# B&R Automation Studio project A2019059_Linka_Power_CP (part 20)

#### Main.st - Init, cyclic, exit code
```iecst
PROGRAM _INIT
    TprazdnyZasobnik.PT:=T#2000ms;
    TakumulaciaPlna.PT:=T#1000ms;
    TvytvorenieVakua.PT:=T#200ms;
    TodvetranieVakua.PT:=T#1s;
    TprefukPredBrzdou.PT:=T#2000ms;
    TprefukZaBrzdou.PT:=T#2000ms;
    TvysuvanieSpindle.PT:=T#1s;
    TpripravaSkrutky.PT:=T#3000ms;
    ToddelovacZakladnaPoloha.PT:=T#1000ms;
    TodsatieNecistot.PT:=T#1000ms;
    Tvibrovanie.PT:=T#3000ms;
    TvyfukovaniePredVibrovanim.PT:= T#1000ms;
    TpodaniaSkrutky.PT:= T#1000ms;
    TpredSkrutkaPripravena.PT:= T#500ms;
    TvypnutieOfuku.PT:= T#2000ms;
    TalarmuVysunutiaSkrutkovacky.PT:= T#10s;
END_PROGRAM

PROGRAM _CYCLIC

	(********************Mapovanie IN/OUT********************************)

    SkrutkovaciSet.Manual:= P1_Srobovanie.SkrutkovaciSet_K30.Manual;
    SkrutkovaciSet.Automat:= P1_Srobovanie.SkrutkovaciSet_K30.Automat;
    SkrutkovaciSet.SkrutkaOdobrata:=P1_Srobovanie.SkrutkovaciSet_K30.SkrutkaK30_Odobrata;
    P1_Srobovanie.SkrutkovaciSet_K30.SkrutkaK30_Pripravena:= SkrutkovaciSet.SkrutkaPripravena;
    P1_Srobovanie.SkrutkovaciSet_K30.CistenieUkoncene:= SkrutkovaciSet.CistenieVykonane;
    SkrutkovaciSet.VykonajCistenie:= P1_Srobovanie.SkrutkovaciSet_K30.Cistenie;

    SkrutkovaciSet.Vreteno.IN.BrakeClosed:=P1_Srobovanie.IN.SkrutkK30_Cist_BrzdaZatvor_MS22;
    SkrutkovaciSet.Vreteno.IN.BrakeOpen:=P1_Srobovanie.IN.SkrutkK30_Cist_BrzdaOtvoren_MS21;
    SkrutkovaciSet.Vreteno.IN.DeptControl:=P1_Srobovanie.IN.SkrutkK30_ZASUNUTY_MS20;
    SkrutkovaciSet.Vreteno.IN.ScrewMeasurement:=P1_Srobovanie.IN.SkrutkK30_SrobaPresla_IS51;
    SkrutkovaciSet.Vreteno.IN.ScrewMeasurementBrake:=P1_Srobovanie.IN.SkrutkK30_Cist_SrobaPresla_IS52;

    IF P1_Srobovanie.SkrutkovaciSet_K30.Reset AND SkrutkovaciSet.VretenoFaza <> 102 AND SkrutkovaciSet.VretenoFaza <> 104 THEN
        SkrutkovaciSet.VretenoFaza:=0;
        P1_Srobovanie.SkrutkovaciSet_K30.Reset:= FALSE;
    END_IF

    SkrutkovaciSet.Zasobnik.IN.AccumulationSwitch:=P1_Srobovanie.IN.ZasobSrobK30_ListaPLNA_OS7;
    SkrutkovaciSet.Zasobnik.IN.FeederLevelControl:=P1_Srobovanie.IN.ZasobSrobK30_PRAZDNY_IS49;
    SkrutkovaciSet.Zasobnik.IN.ScrewMeasurement:=P1_Srobovanie.IN.NastrelSrobK30_SrobaPresla_IS50;

    P1_Srobovanie.OUT.SkrutkK30_Cist_POSUN_YV123:=SkrutkovaciSet.Vreteno.OUT.BlastAirBrake;
    P1_Srobovanie.OUT.SkrutkK30_Cist_OTVOR_YV92:=SkrutkovaciSet.Vreteno.OUT.BrakeSpindle;
    P1_Srobovanie.OUT.SkrutkK30_OfukVakua_RUN_YV91:=SkrutkovaciSet.Vreteno.OUT.CounterBlast;
    IF SkrutkovaciSet.VretenoFaza>1 AND SkrutkovaciSet.VretenoFaza<100 THEN
        P1_Srobovanie.OUT.SkrutkK30_VYSUN_YV89:=SkrutkovaciSet.Vreteno.OUT.Spindle;
    END_IF
    P1_Srobovanie.OUT.SkrutkK30_Cist_ODSAVANIE_YV93:=SkrutkovaciSet.Vreteno.OUT.WasteExtraction;
    IF SkrutkovaciSet.VykonajCistenie THEN
        P1_Srobovanie.OUT.SkrutkK30_PrisavSkrutky_RUN_YV90:=SkrutkovaciSet.Vreteno.OUT.Vacuum;
    END_IF
    P1_Srobovanie.OUT.ZasobSrobK30_Ofuk_RUN_YV85:=SkrutkovaciSet.Zasobnik.OUT.BlowOff;
    P1_Srobovanie.OUT.NastrelSrobK30_PosunSrobu_YV87:=SkrutkovaciSet.Zasobnik.OUT.Escapement;
    P1_Srobovanie.OUT.NastrelSrobK30_NastrelSrobu_YV88:=SkrutkovaciSet.Zasobnik.OUT.FeedAir;
    P1_Srobovanie.OUT.ZasobSrobK30_OfukTried_RUN_YV86:=SkrutkovaciSet.Zasobnik.OUT.SortingAir;
    P1_Srobovanie.OUT.ZasobSrobK30_Vibrovanie_RUN_FM8:= SkrutkovaciSet.Zasobnik.OUT.StartA20;
    (********************Časáky********************************)
    TprazdnyZasobnik();
    TakumulaciaPlna();
    TvytvorenieVakua();
    TodvetranieVakua();
    TprefukPredBrzdou();
    TprefukZaBrzdou();
    TvysuvanieSpindle();
    TpripravaSkrutky();
    ToddelovacZakladnaPoloha();
    TodsatieNecistot();
    Tvibrovanie();
    TvyfukovaniePredVibrovanim();
    TpodaniaSkrutky();
    TpredSkrutkaPripravena();
    TvypnutieOfuku();
    TalarmuVysunutiaSkrutkovacky();
    (********************Zásobnik********************************)

    //kontrola akumulacie
    IF SkrutkovaciSet.Zasobnik.IN.AccumulationSwitch=1 THEN
        TakumulaciaPlna.IN:=1;
    ELSE
        TakumulaciaPlna.IN:=0;
    END_IF

    //kontrola naplnenia zasobnika
    IF SkrutkovaciSet.Zasobnik.IN.FeederLevelControl=1 THEN
        TprazdnyZasobnik.IN:=1;
    ELSE
        TprazdnyZasobnik.IN:=0;
    END_IF

    //Ovládanie vzduchov zásobníka//
    IF ZapniHrniec THEN
        IF TakumulaciaPlna.Q=1 THEN
            SkrutkovaciSet.Zasobnik.OUT.BlowOff:=1;
        ELSE
            SkrutkovaciSet.Zasobnik.OUT.BlowOff:=0;
        END_IF
        SkrutkovaciSet.Zasobnik.OUT.SortingAir:= 1;
    ELSE
        SkrutkovaciSet.Zasobnik.OUT.BlowOff:=0;
    END_IF

    IF NOT SkrutkovaciSet.Zasobnik.OUT.StartA20 AND NOT ZapniHrniec THEN
        TvypnutieOfuku.IN:= 1;
    ELSE
        TvypnutieOfuku.IN:= 0;
    END_IF

    IF EDGEPOS(TvypnutieOfuku.Q) THEN
        SkrutkovaciSet.Zasobnik.OUT.SortingAir:= 0;
    END_IF

    //ovladanie vibracneho podavaca
    IF ZapniHrniec THEN
        TvyfukovaniePredVibrovanim.IN:= 1;
    ELSE
        TvyfukovaniePredVibrovanim.IN:= 0;
    END_IF

    IF ZapniHrniec AND TvyfukovaniePredVibrovanim.Q THEN
        SkrutkovaciSet.Zasobnik.OUT.StartA20:=1;
        Tvibrovanie.IN:=1;
    ELSE
        SkrutkovaciSet.Zasobnik.OUT.StartA20:=0;
        Tvibrovanie.IN:=0;
    END_IF

    IF Tvibrovanie.Q=1 AND NOT P1_Srobovanie.RR_ZapniHrniec_K30 THEN
        IF TakumulaciaPlna.Q=1 THEN
            ZapniHrniec:= 0;
        END_IF
    END_IF

    //Zapnutie hrnca v ručnom režime//
    IF EDGEPOS(P1_Srobovanie.RR_ZapniHrniec_K30) THEN
        ZapniHrniec:= TRUE;
    END_IF
    IF EDGENEG(P1_Srobovanie.RR_ZapniHrniec_K30) THEN
        ZapniHrniec:= FALSE;
    END_IF

    //Zrušenie signálu skrutka pripravená//
    IF SkrutkovaciSet.SkrutkaPripravena=1 THEN
        IF SkrutkovaciSet.SkrutkaOdobrata=1 THEN
            SkrutkovaciSet.SkrutkaPripravena:=0;
        END_IF
    END_IF

    (********************Vreteno********************************)
    CASE SkrutkovaciSet.VretenoFaza OF
        0: SkrutkovaciSet.VretenoStatus:="Vypnute";
            SkrutkovaciSet.Vreteno.OUT.BlastAirBrake:=0;
            SkrutkovaciSet.Vreteno.OUT.BrakeSpindle:=0;
            SkrutkovaciSet.Vreteno.OUT.CounterBlast:=0;
            SkrutkovaciSet.Vreteno.OUT.Spindle:=0;
            SkrutkovaciSet.Vreteno.OUT.Vacuum:=0;
            SkrutkovaciSet.Vreteno.OUT.WasteExtraction:=0;

            SkrutkovaciSet.Zasobnik.OUT.Escapement:=0;
            SkrutkovaciSet.Zasobnik.OUT.FeedAir:=0;
            SkrutkovaciSet.Zasobnik.OUT.StartA20:=0;

            SkrutkovaciSet.CistenieVykonane:=0;
            SkrutkovaciSet.SkrutkaPripravena:=0;

            TprazdnyZasobnik.IN:=0;
            TakumulaciaPlna.IN:=0;
            TvytvorenieVakua.IN:=0;
            TodvetranieVakua.IN:=0;
            TprefukPredBrzdou.IN:=0;
            TprefukZaBrzdou.IN:=0;
            TvysuvanieSpindle.IN:=0;
            TpripravaSkrutky.IN:=0;
            ToddelovacZakladnaPoloha.IN:=0;
            TodsatieNecistot.IN:=0;
            TpodaniaSkrutky.IN:= 0;
            TpredSkrutkaPripravena.IN:= 0;
            TalarmuVysunutiaSkrutkovacky.IN:= 0;
            ZapniHrniec:= 0;
            PocetPokusovOpripravuSkrutky:=0;
            StavSkrutkovackaVysunuta:= 0;
            SkrutkovaciSet.VretenoFaza:=1;

        1: SkrutkovaciSet.VretenoStatus:="Inicializacia: cakam na povel";
            IF SkrutkovaciSet.Automat=1 THEN
                SkrutkovaciSet.CistenieVykonane:=0;
                SkrutkovaciSet.SkrutkaPripravena:=0;
                SkrutkovaciSet.VretenoFaza:=2;
            ELSIF SkrutkovaciSet.Manual=1 THEN
                SkrutkovaciSet.VretenoFaza:=250;
            END_IF

        2: SkrutkovaciSet.VretenoStatus:="Inicializacia: cakam na povel precisti hadice";
            IF SkrutkovaciSet.VykonajCistenie=1 THEN
                SkrutkovaciSet.Vreteno.OUT.Vacuum:=1;
                SkrutkovaciSet.VretenoFaza:=3;
            END_IF

        3: SkrutkovaciSet.VretenoStatus:="Inicializacia: Cakam na snimac: vreteno vysunute";
            SkrutkovaciSet.Vreteno.OUT.Spindle:=1;
            TalarmuVysunutiaSkrutkovacky.IN:= 1;

            IF P1_Srobovanie.IN.SkrutkK30_VysunutieHrotu_IOS8 > 1 THEN
                StavSkrutkovackaVysunuta:= TRUE;
                TvysuvanieSpindle.IN:=1;
            END_IF

            IF TvysuvanieSpindle.Q=1 AND StavSkrutkovackaVysunuta THEN
                TodvetranieVakua.IN:= 1;
                SkrutkovaciSet.Vreteno.OUT.CounterBlast:=1;
                SkrutkovaciSet.Vreteno.OUT.Vacuum:=0;
            END_IF

            IF TvysuvanieSpindle.Q AND StavSkrutkovackaVysunuta AND TodvetranieVakua.Q THEN
                StavSkrutkovackaVysunuta:= FALSE;
                TalarmuVysunutiaSkrutkovacky.IN:= 0;
                TvysuvanieSpindle.IN:=0;
                TodvetranieVakua.IN:= 0;
                SkrutkovaciSet.VretenoFaza:=4;
            ELSIF TalarmuVysunutiaSkrutkovacky.Q THEN
                P1_Alarmy[142]:= TRUE;
                P1_PoruchaST2:= TRUE;
            END_IF

        4: SkrutkovaciSet.VretenoStatus:="Inicializacia: Cakam na snimac: vreteno zasunute";
            SkrutkovaciSet.Vreteno.OUT.Spindle:=0;
            IF SkrutkovaciSet.Vreteno.IN.DeptControl=1 THEN
                SkrutkovaciSet.Vreteno.OUT.CounterBlast:=0;
                SkrutkovaciSet.VretenoFaza:=5;
            END_IF

        5: SkrutkovaciSet.VretenoStatus:="Inicializacia: Cakam na prefuknutie hadice za brzdou";
            TprefukZaBrzdou.IN:=1;
            SkrutkovaciSet.Vreteno.OUT.BlastAirBrake:=1;
            IF TprefukZaBrzdou.Q=1 THEN
                TprefukZaBrzdou.IN:=0;
                SkrutkovaciSet.Vreteno.OUT.BlastAirBrake:=0;
                SkrutkovaciSet.VretenoFaza:=6;
            END_IF

        6: SkrutkovaciSet.VretenoStatus:="Inicializacia: vypinam prefuk";
            TprefukZaBrzdou.IN:=0;
            SkrutkovaciSet.Vreteno.OUT.BlastAirBrake:=0;
            SkrutkovaciSet.Vreteno.OUT.Vacuum:=1;
            SkrutkovaciSet.VretenoFaza:=7;

        7: SkrutkovaciSet.VretenoStatus:="Inicializacia: Cakam na snimac: vreteno vysunute";
            SkrutkovaciSet.Vreteno.OUT.Spindle:=1;
            TalarmuVysunutiaSkrutkovacky.IN:= 1;

            IF P1_Srobovanie.IN.SkrutkK30_VysunutieHrotu_IOS8 > 1 THEN
                StavSkrutkovackaVysunuta:= TRUE;
                TvysuvanieSpindle.IN:=1;
            END_IF

            IF TvysuvanieSpindle.Q=1 AND StavSkrutkovackaVysunuta THEN
                TodvetranieVakua.IN:= 1;
                SkrutkovaciSet.Vreteno.OUT.CounterBlast:=1;
                SkrutkovaciSet.Vreteno.OUT.Vacuum:=0;
            END_IF

            IF TvysuvanieSpindle.Q AND StavSkrutkovackaVysunuta AND TodvetranieVakua.Q THEN
                StavSkrutkovackaVysunuta:= FALSE;
                TalarmuVysunutiaSkrutkovacky.IN:= 0;
                TvysuvanieSpindle.IN:=0;
                TodvetranieVakua.IN:= 0;
                SkrutkovaciSet.VretenoFaza:=8;
            ELSIF TalarmuVysunutiaSkrutkovacky.Q THEN
                P1_Alarmy[142]:= TRUE;
                P1_PoruchaST2:= TRUE;
            END_IF

        8: SkrutkovaciSet.VretenoStatus:="Inicializacia: Cakam na snimac: vreteno zasunute";
            SkrutkovaciSet.Vreteno.OUT.Spindle:=0;
            IF SkrutkovaciSet.Vreteno.IN.DeptControl=1 THEN
                SkrutkovaciSet.Vreteno.OUT.CounterBlast:=0;
                SkrutkovaciSet.VretenoFaza:=9;
            END_IF

        9: SkrutkovaciSet.VretenoStatus:="Inicializacia: Cakam na prefuknutie hadice pred brzdou";
            TprefukPredBrzdou.IN:=1;
            SkrutkovaciSet.Zasobnik.OUT.FeedAir:=1;
            IF TprefukPredBrzdou.Q=1 THEN
                TprefukPredBrzdou.IN:=0;
                SkrutkovaciSet.Zasobnik.OUT.FeedAir:=0;
                SkrutkovaciSet.VretenoFaza:=10;
            END_IF

        10: SkrutkovaciSet.VretenoStatus:="Inicializacia: Cakam na snimac: brzda uvolnena";
            SkrutkovaciSet.Vreteno.OUT.BrakeSpindle:=1;
            IF SkrutkovaciSet.Vreteno.IN.BrakeOpen=1 THEN
                SkrutkovaciSet.Vreteno.OUT.BlastAirBrake:=1;
                SkrutkovaciSet.VretenoFaza:=11;
            END_IF

        11: SkrutkovaciSet.VretenoStatus:="Inicializacia: Cakam na prefuknutie hadice za brzdou";
            TprefukZaBrzdou.IN:=1;
            SkrutkovaciSet.Vreteno.OUT.BlastAirBrake:=1;
            IF TprefukZaBrzdou.Q=1 THEN
                TprefukZaBrzdou.IN:=0;
                SkrutkovaciSet.Vreteno.OUT.BlastAirBrake:=0;
                SkrutkovaciSet.VretenoFaza:=12;
            END_IF

        12: SkrutkovaciSet.VretenoStatus:="Inicializacia: vypinam prefuk";
            TprefukZaBrzdou.IN:=0;
            SkrutkovaciSet.Vreteno.OUT.BlastAirBrake:=0;
            SkrutkovaciSet.Vreteno.OUT.Vacuum:=1;
            SkrutkovaciSet.VretenoFaza:=13;

        13: SkrutkovaciSet.VretenoStatus:="Inicializacia: Cakam na snimac: vreteno vysunute";
            SkrutkovaciSet.Vreteno.OUT.Spindle:=1;
            TalarmuVysunutiaSkrutkovacky.IN:= 1;

            IF P1_Srobovanie.IN.SkrutkK30_VysunutieHrotu_IOS8 > 1 THEN
                StavSkrutkovackaVysunuta:= TRUE;
                TvysuvanieSpindle.IN:=1;
            END_IF

            IF TvysuvanieSpindle.Q=1 AND StavSkrutkovackaVysunuta THEN
                TodvetranieVakua.IN:= 1;
                SkrutkovaciSet.Vreteno.OUT.CounterBlast:=1;
                SkrutkovaciSet.Vreteno.OUT.Vacuum:=0;
            END_IF

            IF TvysuvanieSpindle.Q AND StavSkrutkovackaVysunuta AND TodvetranieVakua.Q THEN
                StavSkrutkovackaVysunuta:= FALSE;
                TalarmuVysunutiaSkrutkovacky.IN:= 0;
                TvysuvanieSpindle.IN:=0;
                TodvetranieVakua.IN:= 0;
                SkrutkovaciSet.VretenoFaza:=14;
            ELSIF TalarmuVysunutiaSkrutkovacky.Q THEN
                P1_Alarmy[142]:= TRUE;
                P1_PoruchaST2:= TRUE;
            END_IF

        14: SkrutkovaciSet.VretenoStatus:="Inicializacia: Cakam na snimac: vreteno zasunute";
            SkrutkovaciSet.Vreteno.OUT.Spindle:=0;
            IF SkrutkovaciSet.Vreteno.IN.DeptControl=1 THEN
                SkrutkovaciSet.Vreteno.OUT.CounterBlast:=0;
                SkrutkovaciSet.VretenoFaza:=15;
            END_IF

        15: SkrutkovaciSet.VretenoStatus:="Inicializacia: Cakam na snimac: brzda zasunuta";
            SkrutkovaciSet.Vreteno.OUT.BrakeSpindle:=0;
            IF SkrutkovaciSet.Vreteno.IN.BrakeClosed=1 THEN
                SkrutkovaciSet.CistenieVykonane:=1;
                SkrutkovaciSet.VretenoFaza:=16;
            END_IF

        16: SkrutkovaciSet.VretenoStatus:="Inicializacia: Cakam na zrusenie signalu: vykonaj cistenie";
            IF SkrutkovaciSet.VykonajCistenie=0 THEN
                SkrutkovaciSet.CistenieVykonane:=0;
                SkrutkovaciSet.SkrutkaPripravena:=0;
                SkrutkovaciSet.VretenoFaza:=100;
            END_IF

        100: SkrutkovaciSet.VretenoStatus:="Cakam kym zasobnik pripravy skrutku";
            ZapniHrniec:= 1;
            IF TakumulaciaPlna.Q=1 AND SkrutkovaciSet.Zasobnik.OUT.StartA20 THEN
                TpodaniaSkrutky.IN:= 1;
            END_IF

            IF TpodaniaSkrutky.Q THEN
                TpodaniaSkrutky.IN:= 0;
                SkrutkovaciSet.VretenoFaza:=102;
            END_IF

        102: SkrutkovaciSet.VretenoStatus:="Cakam na snimac: skrutka presla hadicou";
            SkrutkovaciSet.Zasobnik.OUT.Escapement:=1;
            TpripravaSkrutky.IN:=1;
            IF SkrutkovaciSet.Zasobnik.IN.ScrewMeasurement=1 THEN
                SkrutkovaciSet.Zasobnik.OUT.FeedAir:=1;
                TpripravaSkrutky.IN:=0;
                SkrutkovaciSet.VretenoFaza:=104;
            ELSIF TpripravaSkrutky.Q=1 THEN
                TpripravaSkrutky.IN:=0;
                SkrutkovaciSet.Zasobnik.OUT.Escapement:=0;
                SkrutkovaciSet.VretenoFaza:=100;
            END_IF

        104: SkrutkovaciSet.VretenoStatus:="Cakam na snimac: skrutka presla hadicou pred brzdou";
            IF SkrutkovaciSet.Vreteno.IN.ScrewMeasurementBrake=1 THEN
                SkrutkovaciSet.Zasobnik.OUT.Escapement:=0;
                SkrutkovaciSet.Zasobnik.OUT.FeedAir:=0;
                PocetPokusovOpripravuSkrutky:=0;
                SkrutkovaciSet.VretenoFaza:=106;
            END_IF

        106: SkrutkovaciSet.VretenoStatus:="Cakam na odsatie necistot";
            SkrutkovaciSet.Vreteno.OUT.WasteExtraction:=1;
            TodsatieNecistot.IN:=1;

            IF TodsatieNecistot.Q=1 THEN
                TodsatieNecistot.IN:=0;
                SkrutkovaciSet.Vreteno.OUT.WasteExtraction:=0;
                SkrutkovaciSet.VretenoFaza:=107;
            END_IF

        107: SkrutkovaciSet.VretenoStatus:="Cakam kym skrutkovacka odoberie skrutku";
            IF SkrutkovaciSet.SkrutkaPripravena=0 AND SkrutkovaciSet.SkrutkaOdobrata=0 THEN
                SkrutkovaciSet.VretenoFaza:=108;
            END_IF

        108: SkrutkovaciSet.VretenoStatus:="Cakam na snimac: brzda uvolnena";
            SkrutkovaciSet.Vreteno.OUT.BrakeSpindle:=1;
            IF SkrutkovaciSet.Vreteno.IN.BrakeOpen=1 THEN
                SkrutkovaciSet.Vreteno.OUT.BlastAirBrake:=1;
                SkrutkovaciSet.VretenoFaza:=110;
            END_IF

        110: SkrutkovaciSet.VretenoStatus:="Cakam na snimac: skrutka presla hadicou pred vretenom";
            IF SkrutkovaciSet.Vreteno.IN.ScrewMeasurement=1 THEN
                SkrutkovaciSet.Vreteno.OUT.BlastAirBrake:=0;
                SkrutkovaciSet.Vreteno.OUT.BrakeSpindle:=0;
                SkrutkovaciSet.VretenoFaza:=112;
            END_IF

        112: SkrutkovaciSet.VretenoStatus:="Cakam na snimac: brzda zabrzdena";
            SkrutkovaciSet.Vreteno.OUT.BrakeSpindle:=0;
            IF SkrutkovaciSet.Vreteno.IN.BrakeClosed=1 AND SkrutkovaciSet.SkrutkaOdobrata=0 THEN
                TpredSkrutkaPripravena.IN:= 1;
                IF TpredSkrutkaPripravena.Q THEN
                    TpredSkrutkaPripravena.IN:= 0;
                    SkrutkovaciSet.SkrutkaPripravena:=1;
                    SkrutkovaciSet.VretenoFaza:=100;
                END_IF
            END_IF

            //*************** opakovany pokus o oddelenie skrutky *********************************

        170: SkrutkovaciSet.VretenoStatus:="Cakam na presunutie oddelovaca do zakladnej polohy";
            SkrutkovaciSet.Zasobnik.OUT.Escapement:=0;
            ToddelovacZakladnaPoloha.IN:=1;
            IF ToddelovacZakladnaPoloha.Q=1 THEN
                ToddelovacZakladnaPoloha.IN:=0;
                PocetPokusovOpripravuSkrutky:=PocetPokusovOpripravuSkrutky+1;
                IF PocetPokusovOpripravuSkrutky>3 THEN
                    PocetPokusovOpripravuSkrutky:=0;
                    SkrutkovaciSet.VretenoFaza:=171;
                ELSE
                    SkrutkovaciSet.VretenoFaza:=100;
                END_IF
            END_IF

        171: SkrutkovaciSet.VretenoStatus:="Zaseknuta skrutka v oddelovaci!!!";

    END_CASE
END_PROGRAM

PROGRAM _EXIT
END_PROGRAM
```

#### Types.typ - Local data types
```iecst
(*skrutkovacka M5x55 P2*)

TYPE
	SkrutkovaciSetStruc : 	STRUCT
		VretenoStatus : WSTRING[80];
		VretenoFaza : USINT;
		Zasobnik : ZasobnikStruc;
		Vreteno : VretenoStruc;
		SkrutkaOdobrata : BOOL;
		SkrutkaPripravena : BOOL;
		Manual : BOOL;
		PodajSrobu : BOOL;
		CistenieVykonane : BOOL;
		VykonajCistenie : BOOL;
		Automat : BOOL;
	END_STRUCT;
	INzasobnik : 	STRUCT
		AccumulationSwitch : BOOL; (*Snimac zaplnenia S25*)
		ScrewMeasurement : BOOL; (*Kontrola matice S21*)
		FeederLevelControl : BOOL; (*Hladina v zasobniku S20*)
	END_STRUCT;
	OUTzasobnik : 	STRUCT
		StartA20 : BOOL; (*Zapnutie vibrovania A20*)
		Escapement : BOOL; (*Pustanie matky do hadice Y22*)
		FeedAir : BOOL; (*Strielanie do hadice Y21*)
		SortingAir : BOOL; (*Triedenie kusov Y30*)
		BlowOff : BOOL; (*Zhadzovanie kusov Y25*)
	END_STRUCT;
	INvreteno : 	STRUCT
		ReturnStroke : BOOL; (*Vreteno zasunute S01*)
		DeptControl : BOOL; (*Vreteno vysunute S02*)
		BrakeClosed : BOOL; (*Brzda zatvorena S13*)
		BrakeOpen : BOOL; (*Brzda otvorena S12*)
		ScrewMeasurementBrake : BOOL; (*Kontrola matice pred brzdou S15*)
		ScrewMeasurement : BOOL; (*Kontrola matice v hadici S06*)
	END_STRUCT;
	OUTvreteno : 	STRUCT
		WasteExtraction : BOOL; (*Odstranovanie spiny Y13*)
		Spindle : BOOL; (*Vysunutie vretena Y02*)
		BlastAirBrake : BOOL; (*Strielanie za brzdou Y14*)
		BrakeSpindle : BOOL; (*Brzda vretena Y12*)
		Vacuum : BOOL; (*Pridrzanie skrutky Y15*)
		CounterBlast : BOOL; (*Uvolnenie skrutky Y16*)
	END_STRUCT;
	VretenoStruc : 	STRUCT
		OUT : OUTvreteno;
		IN : INvreteno;
	END_STRUCT;
	ZasobnikStruc : 	STRUCT
		OUT : OUTzasobnik;
		IN : INzasobnik;
	END_STRUCT;
END_TYPE
```

#### Variables.var - Local variables
```iecst
VAR
	SkrutkovaciSet : SkrutkovaciSetStruc;
	TprazdnyZasobnik : TON;
	TakumulaciaPlna : TON;
	TvytvorenieVakua : TON;
	TodvetranieVakua : TON;
	TprefukPredBrzdou : TON;
	TvysuvanieSpindle : TON;
	TprefukZaBrzdou : TON;
	PocetPokusovOpripravuSkrutky : USINT;
	ToddelovacZakladnaPoloha : TON;
	TpripravaSkrutky : TON;
	TodsatieNecistot : TON;
	Tvibrovanie : TON;
	TvyfukovaniePredVibrovanim : TON;
	ZapniHrniec : BOOL;
	TpodaniaSkrutky : TON;
	TpredSkrutkaPripravena : TON;
	TvypnutieOfuku : TON;
	StavSkrutkovackaVysunuta : BOOL;
	TalarmuVysunutiaSkrutkovacky : TON;
END_VAR
```

### Program Logical/Program/Pracovisko_1/P1_SkrutkovaciSet_M5 (IEC)

#### Main.st - Init, cyclic, exit code
```iecst
PROGRAM _INIT
	TprazdnyZasobnik.PT:=T#2000ms;
	TakumulaciaPlna.PT:=T#1000ms;
	TakumulaciaPrazdna.PT:=T#1000ms;
	TvytvorenieVakua.PT:=T#200ms;
	TodvetranieVakua.PT:=T#200ms;
	TvibrovanieHrniec.PT:=T#3000ms;
	TvibrovanieLista.PT:=T#5000ms;
	TpredOtocenim.PT:= T#1000ms;
	TvyfukovaniePredVibrovanim.PT:= T#1000ms;
	TpodaniaSkrutky.PT:= T#1000ms;
	TvypnutieOfuku.PT:= T#2000ms;
	TpoOtoceni.PT:= T#5s;
	TofukVibrolisty.PT:= T#1000ms;
END_PROGRAM

PROGRAM _CYCLIC

	(********************Mapovanie IN/OUT********************************)
	SkrutkovaciSet.Manual:= P1_Srobovanie.SkrutkovaciSet_M5.Manual;
	SkrutkovaciSet.Automat:= P1_Srobovanie.SkrutkovaciSet_M5.Automat;
	SkrutkovaciSet.SkrutkaOdobrata:=P1_Srobovanie.SkrutkovaciSet_M5.SkrutkaM5_Odobrata;
	P1_Srobovanie.SkrutkovaciSet_M5.SkrutkaM5_Pripravena:= SkrutkovaciSet.SkrutkaPripravena;

	IF P1_Srobovanie.SkrutkovaciSet_M5.Reset THEN
		SkrutkovaciSet.VretenoFaza:=0;
		P1_Srobovanie.SkrutkovaciSet_M5.Reset:= FALSE;
	END_IF

	SkrutkovaciSet.Vreteno.IN.ReturnStroke:=P1_Srobovanie.IN.SkrutkM5_ZASUNUTY_MS39;
	SkrutkovaciSet.Vreteno.IN.VakuumDosiahnute:=P1_Srobovanie.IN.SkrutkM5_SnimacVakua_S28;

	SkrutkovaciSet.Zasobnik.IN.AccumulationSwitchStart:=P1_Srobovanie.IN.VibrolistaSrobM5_KONIEC_OS9;
	SkrutkovaciSet.Zasobnik.IN.AccumulationSwitchEnd:=P1_Srobovanie.IN.ZasobSrobM5_ListaPLNA_OS8;
	SkrutkovaciSet.Zasobnik.IN.EscapementPickUp:=P1_Srobovanie.IN.OddelSrobM5_OtocenyVZAD_MS38;
	SkrutkovaciSet.Zasobnik.IN.EscapementDrop:=P1_Srobovanie.IN.OddelSrobM5_OtocenyVPRED_MS37;
	SkrutkovaciSet.Zasobnik.IN.FeederLevelControl:=P1_Srobovanie.IN.ZasobSrobM5_PRAZDNY_IS53;
	SkrutkovaciSet.Zasobnik.IN.InlineControl:=P1_Srobovanie.IN.OddelSrobM5_SrobaNaVstupe_OS13;
	SkrutkovaciSet.Zasobnik.IN.ScrewAvailable:=P1_Srobovanie.IN.OddelSrobM5_SrobaNaVystupe_OS14;

	P1_Srobovanie.OUT.ZasobSrobM5_Ofuk_RUN_YV94:=SkrutkovaciSet.Zasobnik.OUT.BlowOff;
	P1_Srobovanie.OUT.OddelovacSrobM5_OtocVPRED_YV103:=SkrutkovaciSet.Zasobnik.OUT.EscapementDrop;
	P1_Srobovanie.OUT.OddelovacSrobM5_OtocVZAD_YV102:=SkrutkovaciSet.Zasobnik.OUT.EscapementPickUp;
	P1_Srobovanie.OUT.ZasobSrobM5_OfukTried_RUN_YV95:=SkrutkovaciSet.Zasobnik.OUT.SortingAir;
	P1_Srobovanie.OUT.ZasobSrobM5_Vibrov_RUN_FM10:=SkrutkovaciSet.Zasobnik.OUT.StartA20Hrniec;
	P1_Srobovanie.OUT.VibrolistaSrobM5_Vibrov_RUN_FM11:=SkrutkovaciSet.Zasobnik.OUT.StartA20Lista;

	(********************Časáky********************************)
	TprazdnyZasobnik();
	TakumulaciaPlna();
	TakumulaciaPrazdna();
	TvytvorenieVakua();
	TodvetranieVakua();
	TvibrovanieHrniec();
	TvibrovanieLista();
	TpredOtocenim();
	TvyfukovaniePredVibrovanim();
	TpodaniaSkrutky();
	TvypnutieOfuku();
	TpoOtoceni();
	TofukVibrolisty();
	(********************Zásobnik********************************)
	//kontrola akumulacie
	IF SkrutkovaciSet.Zasobnik.IN.AccumulationSwitchStart=1 THEN
		TakumulaciaPlna.IN:=1;
	ELSE
		TakumulaciaPlna.IN:=0;
	END_IF

	IF SkrutkovaciSet.Zasobnik.IN.AccumulationSwitchEnd=0 THEN
		TakumulaciaPrazdna.IN:=1;
	ELSE
		TakumulaciaPrazdna.IN:=0;
	END_IF

	//kontrola naplnenia zasobnika
	IF SkrutkovaciSet.Zasobnik.IN.FeederLevelControl=1 THEN
		TprazdnyZasobnik.IN:=1;
	ELSE
		TprazdnyZasobnik.IN:=0;
	END_IF

	//Ovládanie vzduchov zásobníka//
	IF ZapniHrniec THEN
		IF TakumulaciaPlna.Q=1 AND TakumulaciaPrazdna.Q=0  THEN
			SkrutkovaciSet.Zasobnik.OUT.BlowOff:=1;
		ELSIF TakumulaciaPrazdna.Q=1 THEN
			SkrutkovaciSet.Zasobnik.OUT.BlowOff:=0;
		END_IF
		SkrutkovaciSet.Zasobnik.OUT.SortingAir:= 1;
	ELSIF ZapniListu THEN
		TofukVibrolisty.IN:= TRUE;
		SkrutkovaciSet.Zasobnik.OUT.SortingAir:= NOT TofukVibrolisty.Q;
	ELSE
		SkrutkovaciSet.Zasobnik.OUT.BlowOff:=0;
	END_IF

	TvypnutieOfuku.IN:= NOT SkrutkovaciSet.Zasobnik.OUT.StartA20Hrniec;

	IF TvypnutieOfuku.Q THEN
		SkrutkovaciSet.Zasobnik.OUT.SortingAir:= 0;
	END_IF

	//ovladanie vibracneho podavaca
	IF SkrutkovaciSet.VretenoFaza>3 AND SkrutkovaciSet.VretenoFaza<250 THEN
		IF SkrutkovaciSet.Zasobnik.IN.AccumulationSwitchStart=0 THEN
			ZapniHrniec:=1;
		ELSIF TvibrovanieHrniec.Q=1 AND SkrutkovaciSet.Zasobnik.IN.AccumulationSwitchEnd=1 AND NOT P1_Srobovanie.RR_ZapniHrniec_M5 THEN
			ZapniHrniec:=0;
		END_IF
	END_IF

	IF ZapniHrniec THEN
		TvyfukovaniePredVibrovanim.IN:= 1;
	ELSE
		TvyfukovaniePredVibrovanim.IN:= 0;
	END_IF

	IF ZapniHrniec AND TvyfukovaniePredVibrovanim.Q THEN
		ZapniListu:=TRUE;
		SkrutkovaciSet.Zasobnik.OUT.StartA20Hrniec:=1;
	ELSE
		SkrutkovaciSet.Zasobnik.OUT.StartA20Hrniec:=0;
	END_IF

	IF SkrutkovaciSet.Zasobnik.IN.AccumulationSwitchEnd=1 THEN
		TvibrovanieHrniec.IN:=1;
	ELSE
		TvibrovanieHrniec.IN:=0;
	END_IF

	//Ovládanie vybrolišty//
	IF ZapniListu AND TofukVibrolisty.Q THEN
		SkrutkovaciSet.Zasobnik.OUT.StartA20Lista:= TRUE;
	ELSE
		SkrutkovaciSet.Zasobnik.OUT.StartA20Lista:= FALSE;
	END_IF

	IF SkrutkovaciSet.Zasobnik.IN.AccumulationSwitchStart=1 AND SkrutkovaciSet.Zasobnik.OUT.StartA20Lista=1 THEN
		TvibrovanieLista.IN:=1;
	ELSE
		TvibrovanieLista.IN:=0;
	END_IF

	IF TvibrovanieLista.Q AND NOT SkrutkovaciSet.Zasobnik.IN.EscapementPickUp AND NOT P1_Srobovanie.RR_ZapniVibrolistu_M5 AND NOT SkrutkovaciSet.Zasobnik.OUT.StartA20Hrniec THEN
		ZapniListu:= FALSE;
	END_IF

	//Zapnutie hrnca v ručnom režime//
	IF EDGEPOS(P1_Srobovanie.RR_ZapniHrniec_M5) THEN
		ZapniHrniec:= TRUE;
	END_IF
	IF EDGENEG(P1_Srobovanie.RR_ZapniHrniec_M5) THEN
		ZapniHrniec:= FALSE;
	END_IF

	//Zapnutie vybrolisty v ručnom režime//
	IF EDGEPOS(P1_Srobovanie.RR_ZapniVibrolistu_M5) THEN
		ZapniListu:= TRUE;
	END_IF

	IF EDGENEG(P1_Srobovanie.RR_ZapniVibrolistu_M5) THEN
		ZapniListu:= FALSE;
	END_IF

	//Otáčenie podavača v ručnom režime//
	IF P1_Srobovanie.RR_OtocPodavacM5_VPRED THEN
		SkrutkovaciSet.Zasobnik.OUT.EscapementPickUp:= FALSE;
		SkrutkovaciSet.Zasobnik.OUT.EscapementDrop:= TRUE;
		P1_Srobovanie.RR_OtocPodavacM5_VPRED:= FALSE;
	ELSIF P1_Srobovanie.RR_OtocPodavacM5_VZAD THEN
		SkrutkovaciSet.Zasobnik.OUT.EscapementDrop:= FALSE;
		SkrutkovaciSet.Zasobnik.OUT.EscapementPickUp:= TRUE;
		P1_Srobovanie.RR_OtocPodavacM5_VZAD:= FALSE;
	END_IF

	IF P1_Srobovanie.IN.OddelSrobM5_OtocenyVPRED_MS37 THEN
		SkrutkovaciSet.Zasobnik.OUT.EscapementDrop:= FALSE;
	END_IF

	IF P1_Srobovanie.IN.OddelSrobM5_OtocenyVZAD_MS38 THEN
		SkrutkovaciSet.Zasobnik.OUT.EscapementPickUp:= FALSE;
	END_IF

	(********************Vreteno********************************)
	CASE SkrutkovaciSet.VretenoFaza OF
		0: SkrutkovaciSet.VretenoStatus:="Vypnute";
			SkrutkovaciSet.Vreteno.OUT.Spindle:=0;
			SkrutkovaciSet.Vreteno.OUT.VacuumOff:=0;
			SkrutkovaciSet.Vreteno.OUT.VacuumOn:=0;

			SkrutkovaciSet.Zasobnik.OUT.EscapementDrop:=0;
			SkrutkovaciSet.Zasobnik.OUT.EscapementPickUp:=0;
			SkrutkovaciSet.Zasobnik.OUT.StartA20Hrniec:=0;
			SkrutkovaciSet.Zasobnik.OUT.StartA20Lista:=0;
			SkrutkovaciSet.Manual:= 0;
			SkrutkovaciSet.Automat:= 0;
			SkrutkovaciSet.SkrutkaOdobrata:= 0;
			SkrutkovaciSet.SkrutkaPripravena:= 0;
			TpredOtocenim.IN:= 0;
			TpoOtoceni.IN:= 0;
			TvyfukovaniePredVibrovanim.IN:= 0;
			TpodaniaSkrutky.IN:= 0;
			ZapniHrniec:= 0;
			ZapniListu:= 0;
			P1_Srobovanie.STAV.Podanie_M5_BUSY:= FALSE;
			SkrutkovaciSet.VretenoFaza:=1;

		1: SkrutkovaciSet.VretenoStatus:="Inicializacia: cakam na povel";
			IF SkrutkovaciSet.Automat=1 THEN
				SkrutkovaciSet.VretenoFaza:=2;
			ELSIF SkrutkovaciSet.Manual=1 THEN
				SkrutkovaciSet.VretenoFaza:=250;
			ELSIF P1_Srobovanie.RR_PodajSkrutkuM5 THEN
				P1_Srobovanie.STAV.Podanie_M5_BUSY:= TRUE;
				SkrutkovaciSet.VretenoFaza:=2;
			END_IF

		2: SkrutkovaciSet.VretenoStatus:="Inicializacia: Cakam na natocenie kolisky na vstup";
			IF SkrutkovaciSet.Zasobnik.IN.ScrewAvailable=1 THEN
				SkrutkovaciSet.VretenoFaza:=10;
			ELSE
				SkrutkovaciSet.Zasobnik.OUT.EscapementDrop:=0;
				SkrutkovaciSet.Zasobnik.OUT.EscapementPickUp:=1;
				IF SkrutkovaciSet.Zasobnik.IN.EscapementPickUp=1 THEN
					SkrutkovaciSet.VretenoFaza:=3;
				END_IF
			END_IF

		3: SkrutkovaciSet.VretenoStatus:="Inicializacia: Cakam na pritomnost skrutky na vstupe";
			ZapniListu:=1;
			ZapniHrniec:= 1;
			IF SkrutkovaciSet.Zasobnik.IN.InlineControl=1 THEN
				SkrutkovaciSet.VretenoFaza:=4;
			END_IF

		4: SkrutkovaciSet.VretenoStatus:="Inicializacia: Natocenie kolisky na vystup";
			TpredOtocenim.IN:= 1;
			IF TpredOtocenim.Q THEN
				TpredOtocenim.IN:= 0;
				SkrutkovaciSet.Zasobnik.OUT.EscapementDrop:=1;
				SkrutkovaciSet.Zasobnik.OUT.EscapementPickUp:=0;
				SkrutkovaciSet.VretenoFaza:=8;
			END_IF

		8: SkrutkovaciSet.VretenoStatus:="Inicializacia: Cakam na natocenie kolisky na vystup";
			TpoOtoceni.IN:= 1;
			IF SkrutkovaciSet.Zasobnik.IN.EscapementDrop=1 THEN
				TpoOtoceni.IN:= 0;
				SkrutkovaciSet.VretenoFaza:=10;
			ELSIF TpoOtoceni.Q THEN
				TpoOtoceni.IN:= 0;
				SkrutkovaciSet.Zasobnik.OUT.EscapementDrop:=0;
				SkrutkovaciSet.Zasobnik.OUT.EscapementPickUp:=1;
				SkrutkovaciSet.VretenoFaza:=4;
			END_IF

		10: SkrutkovaciSet.VretenoStatus:="Inicializacia: Cakam na pritomnost skrutky na vystupe";
			IF SkrutkovaciSet.Zasobnik.IN.ScrewAvailable=1 THEN
				SkrutkovaciSet.VretenoFaza:=100;
			END_IF

		100: SkrutkovaciSet.VretenoStatus:="Pripravene: cakam na povel";
			SkrutkovaciSet.SkrutkaPripravena:=1;
			IF SkrutkovaciSet.SkrutkaOdobrata=1 THEN
				SkrutkovaciSet.VretenoFaza:=101;
			ELSIF P1_Srobovanie.RR_PodajSkrutkuM5 THEN
				P1_Srobovanie.STAV.Podanie_M5_BUSY:= FALSE;
				P1_Srobovanie.RR_PodajSkrutkuM5:= FALSE;
				SkrutkovaciSet.VretenoFaza:=0;
			END_IF

		101: SkrutkovaciSet.VretenoStatus:="Cakam kym zmizne skrutka zo snimaca";

			IF SkrutkovaciSet.Zasobnik.IN.ScrewAvailable=0 THEN
				SkrutkovaciSet.SkrutkaPripravena:=0;
				SkrutkovaciSet.VretenoFaza:=102;
			END_IF

		102: SkrutkovaciSet.VretenoStatus:="Cakam na zrusenie signalu skrutka odobrata";
			IF SkrutkovaciSet.SkrutkaOdobrata=0 THEN
				SkrutkovaciSet.VretenoFaza:=150;
			END_IF

		150: SkrutkovaciSet.VretenoStatus:="Cakam na otocenie kolisky na vstup";
			SkrutkovaciSet.Zasobnik.OUT.EscapementDrop:=0;
			SkrutkovaciSet.Zasobnik.OUT.EscapementPickUp:=1;
			IF SkrutkovaciSet.Zasobnik.IN.EscapementPickUp=1 THEN
				ZapniListu:=1;
				ZapniHrniec:= 1;
				SkrutkovaciSet.VretenoFaza:=151;
			END_IF

		151: SkrutkovaciSet.VretenoStatus:="Inicializacia: Cakam na pritomnost skrutky na vstupe";
			IF SkrutkovaciSet.Zasobnik.IN.InlineControl=1 THEN
				SkrutkovaciSet.VretenoFaza:=152;
			END_IF

		152: SkrutkovaciSet.VretenoStatus:="Inicializacia: Natocenie kolisky na vystup";
			TpredOtocenim.IN:= 1;
			IF TpredOtocenim.Q THEN
				TpredOtocenim.IN:= 0;
				SkrutkovaciSet.Zasobnik.OUT.EscapementDrop:=1;
				SkrutkovaciSet.Zasobnik.OUT.EscapementPickUp:=0;
				SkrutkovaciSet.VretenoFaza:=153;
			END_IF

		153: SkrutkovaciSet.VretenoStatus:="Inicializacia: Cakam na natocenie kolisky na vystup";
			TpoOtoceni.IN:= 1;
			IF SkrutkovaciSet.Zasobnik.IN.EscapementDrop=1 THEN
				TpoOtoceni.IN:= 0;
				SkrutkovaciSet.VretenoFaza:=155;
			ELSIF TpoOtoceni.Q THEN
				TpoOtoceni.IN:= 0;
				SkrutkovaciSet.Zasobnik.OUT.EscapementDrop:=0;
				SkrutkovaciSet.Zasobnik.OUT.EscapementPickUp:=1;
				SkrutkovaciSet.VretenoFaza:=152;
			END_IF

		155: SkrutkovaciSet.VretenoStatus:="Inicializacia: Cakam na pritomnost skrutky na vystupe";
			IF SkrutkovaciSet.Zasobnik.IN.ScrewAvailable=1 THEN
				SkrutkovaciSet.VretenoFaza:=100;
			END_IF

		250: SkrutkovaciSet.VretenoStatus:="Rucny rezim";
			SkrutkovaciSet.Manual:=0;
	END_CASE

END_PROGRAM

PROGRAM _EXIT
END_PROGRAM
```

#### Types.typ - Local data types
```iecst
TYPE
	SkrutkovaciSetStruc : 	STRUCT
		VretenoStatus : WSTRING[80];
		VretenoFaza : USINT;
		Zasobnik : ZasobnikStruc;
		Vreteno : VretenoStruc;
		SkrutkaOdobrata : BOOL;
		SkrutkaPripravena : BOOL;
		Manual : BOOL;
		Automat : BOOL;
	END_STRUCT;
	INzasobnik : 	STRUCT
		AccumulationSwitchEnd : BOOL; (*Snimac zaplnenia listy koniec S28*)
		AccumulationSwitchStart : BOOL; (*Snimac zaplnenia zaciatok listy S25*)
		EscapementDrop : BOOL; (*Koliska na odoberani skrutky S22*)
		EscapementPickUp : BOOL; (*Koliska na naberani skrutky S23*)
		InlineControl : BOOL; (*Srobka v koliske S24*)
		ScrewAvailable : BOOL; (*Srobka na odoberani S21*)
		FeederLevelControl : BOOL; (*Hladina v zasobniku S20*)
	END_STRUCT;
	OUTzasobnik : 	STRUCT
		StartA20Lista : BOOL; (*Zapnutie vibrovania A20 na liste*)
		StartA20Hrniec : BOOL; (*Zapnutie vibrovania A20 v hrnci*)
		EscapementDrop : BOOL; (*Koliska na odoberanie Y22*)
		EscapementPickUp : BOOL; (*Koliska na naberanie Y23*)
		SortingAir : BOOL; (*Triedenie kusov Y30*)
		BlowOff : BOOL; (*Zhadzovanie kusov Y25*)
	END_STRUCT;
	INvreteno : 	STRUCT
		VretenoVysunuteSrobovanie : BOOL; (*IOlink signal*)
		VretenoVysunuteOdhadzovanie : BOOL; (*IOlink signal*)
		VretenoVysunuteOdoberanie : BOOL; (*IOlink signal*)
		VakuumDosiahnute : BOOL; (*Vakuum dosiahnute S28*)
		ReturnStroke : BOOL; (*Vreteno zasunute S01*)
	END_STRUCT;
	OUTvreteno : 	STRUCT
		Spindle : BOOL; (*Vysunutie vretena Y02*)
		VacuumOff : BOOL; (*Vypnutie vakua na pridrzanie skrutky Y15*)
		VacuumOn : BOOL; (*Pridrzanie skrutky Y15*)
	END_STRUCT;
	VretenoStruc : 	STRUCT
		OUT : OUTvreteno;
		IN : INvreteno;
	END_STRUCT;
	ZasobnikStruc : 	STRUCT
		OUT : OUTzasobnik;
		IN : INzasobnik;
	END_STRUCT;
END_TYPE
```

#### Variables.var - Local variables
```iecst
VAR
	SkrutkovaciSet : SkrutkovaciSetStruc;
	TprazdnyZasobnik : TON;
	TakumulaciaPrazdna : TON;
	TakumulaciaPlna : TON;
	TvytvorenieVakua : TON;
	TodvetranieVakua : TON;
	TvibrovanieLista : TON;
	TvibrovanieHrniec : TON;
	TpredOtocenim : TON;
	TvyfukovaniePredVibrovanim : TON;
	ZapniHrniec : BOOL;
	ZapniListu : BOOL;
	TpodaniaSkrutky : TON;
	TvypnutieOfuku : TON;
	TpoOtoceni : TON;
	TofukVibrolisty : TON;
END_VAR
```

### Program Logical/Program/Pracovisko_1/P1_SkrutkovaciSet_M4 (IEC)

#### Main.st - Init, cyclic, exit code
```iecst
PROGRAM _INIT
    TprazdnyZasobnik.PT:=T#2000ms;
    TakumulaciaPlna.PT:=T#1000ms;
    TvytvorenieVakua.PT:=T#200ms;
    TodvetranieVakua.PT:=T#1s;
    TprefukPredBrzdou.PT:=T#2000ms;
    TprefukZaBrzdou.PT:=T#2000ms;
    TvysuvanieSpindle.PT:=T#1s;
    TpripravaSkrutky.PT:=T#3000ms;
    ToddelovacZakladnaPoloha.PT:=T#1000ms;
    TodsatieNecistot.PT:=T#1000ms;
    Tvibrovanie.PT:=T#3000ms;
    TvyfukovaniePredVibrovanim.PT:= T#1000ms;
    TpodaniaSkrutky.PT:= T#1000ms;
    TpredSkrutkaPripravena.PT:= T#1s;
    TvypnutieOfuku.PT:= T#2000ms;
    TalarmuVysunutiaSkrutkovacky.PT:= T#10s;
END_PROGRAM

PROGRAM _CYCLIC

	(********************Mapovanie IN/OUT********************************)

    SkrutkovaciSet.Manual:= P1_Srobovanie.SkrutkovaciSet_M4.Manual;
    SkrutkovaciSet.Automat:= P1_Srobovanie.SkrutkovaciSet_M4.Automat;
    SkrutkovaciSet.SkrutkaOdobrata:=P1_Srobovanie.SkrutkovaciSet_M4.SkrutkaM4_Odobrata;
    P1_Srobovanie.SkrutkovaciSet_M4.SkrutkaM4_Pripravena:= SkrutkovaciSet.SkrutkaPripravena;
    P1_Srobovanie.SkrutkovaciSet_M4.CistenieUkoncene:= SkrutkovaciSet.CistenieVykonane;
    SkrutkovaciSet.VykonajCistenie:= P1_Srobovanie.SkrutkovaciSet_M4.Cistenie;

    SkrutkovaciSet.Vreteno.IN.BrakeClosed:=P1_Srobovanie.IN.SkrutkM4_Cist_BrzdaZatvoren_MS19;
    SkrutkovaciSet.Vreteno.IN.BrakeOpen:=P1_Srobovanie.IN.SkrutkM4_Cist_BrzdaOtvorena_MS18;
    SkrutkovaciSet.Vreteno.IN.DeptControl:=P1_Srobovanie.IN.SkrutkM4_ZASUNUTY_MS17;
    SkrutkovaciSet.Vreteno.IN.ScrewMeasurement:=P1_Srobovanie.IN.SkrutkM4_SrobaPresla_IS47;
    SkrutkovaciSet.Vreteno.IN.ScrewMeasurementBrake:=P1_Srobovanie.IN.SkrutkM4_Cist_SrobaPresla_IS48;

    IF P1_Srobovanie.SkrutkovaciSet_M4.Reset AND SkrutkovaciSet.VretenoFaza <> 102 AND SkrutkovaciSet.VretenoFaza <> 104 THEN
        SkrutkovaciSet.VretenoFaza:=0;
        P1_Srobovanie.SkrutkovaciSet_M4.Reset:= FALSE;
    END_IF

    SkrutkovaciSet.Zasobnik.IN.AccumulationSwitch:=P1_Srobovanie.IN.ZasobSrobM4_ListaPLNA_OS6;
    SkrutkovaciSet.Zasobnik.IN.FeederLevelControl:=P1_Srobovanie.IN.ZasobSrobM4_PRAZDNY_IS44;
    SkrutkovaciSet.Zasobnik.IN.ScrewMeasurement:=P1_Srobovanie.IN.NastrelSrobM4_SrobaPresla_IS46;

    P1_Srobovanie.OUT.SkrutkM4_Cist_POSUN_YV83:=SkrutkovaciSet.Vreteno.OUT.BlastAirBrake;
    P1_Srobovanie.OUT.SkrutkM4_Cist_OTVOR_YV82:=SkrutkovaciSet.Vreteno.OUT.BrakeSpindle;
    P1_Srobovanie.OUT.SkrutkM4_OfukVakua_RUN_YV80:=SkrutkovaciSet.Vreteno.OUT.CounterBlast;
    IF SkrutkovaciSet.VretenoFaza>1 AND SkrutkovaciSet.VretenoFaza<100 THEN
        P1_Srobovanie.OUT.SkrutkM4_VYSUN_YV79:=SkrutkovaciSet.Vreteno.OUT.Spindle;
    END_IF
    P1_Srobovanie.OUT.SkrutkM4_Cist_ODSAVANIE_YV84:=SkrutkovaciSet.Vreteno.OUT.WasteExtraction;
    IF SkrutkovaciSet.VykonajCistenie THEN
        P1_Srobovanie.OUT.SkrutkM4_PrisavSkrutky_RUN_YV81:=SkrutkovaciSet.Vreteno.OUT.Vacuum;
    END_IF
    P1_Srobovanie.OUT.ZasobSrobM4_Ofuk_RUN_YV72:=SkrutkovaciSet.Zasobnik.OUT.BlowOff;
    P1_Srobovanie.OUT.NastrelSrobM4_PosunSrobu_YV77:=SkrutkovaciSet.Zasobnik.OUT.Escapement;
    P1_Srobovanie.OUT.NastrelSrobM4_NastrelSrobu_YV78:=SkrutkovaciSet.Zasobnik.OUT.FeedAir;
    P1_Srobovanie.OUT.ZasobSrobM4_OfukTried_RUN_YV73:=SkrutkovaciSet.Zasobnik.OUT.SortingAir;
    P1_Srobovanie.OUT.ZasobSrobM4_Vibrovanie_RUN_FM9:= SkrutkovaciSet.Zasobnik.OUT.StartA20;
    (********************Časáky********************************)
    TprazdnyZasobnik();
    TakumulaciaPlna();
    TvytvorenieVakua();
    TodvetranieVakua();
    TprefukPredBrzdou();
    TprefukZaBrzdou();
    TvysuvanieSpindle();
    TpripravaSkrutky();
    ToddelovacZakladnaPoloha();
    TodsatieNecistot();
    Tvibrovanie();
    TvyfukovaniePredVibrovanim();
    TpodaniaSkrutky();
    TpredSkrutkaPripravena();
    TvypnutieOfuku();
    TalarmuVysunutiaSkrutkovacky();
    (********************Zásobnik********************************)

    //kontrola akumulacie
    IF SkrutkovaciSet.Zasobnik.IN.AccumulationSwitch=1 THEN
        TakumulaciaPlna.IN:=1;
    ELSE
        TakumulaciaPlna.IN:=0;
    END_IF

    //kontrola naplnenia zasobnika
    IF SkrutkovaciSet.Zasobnik.IN.FeederLevelControl=1 THEN
        TprazdnyZasobnik.IN:=1;
    ELSE
        TprazdnyZasobnik.IN:=0;
    END_IF

    //Ovládanie vzduchov zásobníka//
    IF ZapniHrniec THEN
        IF TakumulaciaPlna.Q=1 THEN
            SkrutkovaciSet.Zasobnik.OUT.BlowOff:=1;
        ELSE
            SkrutkovaciSet.Zasobnik.OUT.BlowOff:=0;
        END_IF
        SkrutkovaciSet.Zasobnik.OUT.SortingAir:= 1;
    ELSE
        SkrutkovaciSet.Zasobnik.OUT.BlowOff:=0;
    END_IF

    IF NOT SkrutkovaciSet.Zasobnik.OUT.StartA20 AND NOT ZapniHrniec THEN
        TvypnutieOfuku.IN:= 1;
    ELSE
        TvypnutieOfuku.IN:= 0;
    END_IF

    IF EDGEPOS(TvypnutieOfuku.Q) THEN
        SkrutkovaciSet.Zasobnik.OUT.SortingAir:= 0;
    END_IF

    //ovladanie vibracneho podavaca
    IF ZapniHrniec THEN
        TvyfukovaniePredVibrovanim.IN:= 1;
    ELSE
        TvyfukovaniePredVibrovanim.IN:= 0;
    END_IF

    IF ZapniHrniec AND TvyfukovaniePredVibrovanim.Q THEN
        SkrutkovaciSet.Zasobnik.OUT.StartA20:=1;
        Tvibrovanie.IN:=1;
    ELSE
        SkrutkovaciSet.Zasobnik.OUT.StartA20:=0;
        Tvibrovanie.IN:=0;
    END_IF

    IF Tvibrovanie.Q=1 THEN
        IF TakumulaciaPlna.Q=1 AND NOT P1_Srobovanie.RR_ZapniHrniec_M4 THEN
            ZapniHrniec:= 0;
        END_IF
    END_IF

    //Zapnutie hrnca v ručnom režime//
    IF EDGEPOS(P1_Srobovanie.RR_ZapniHrniec_M4) THEN
        ZapniHrniec:= TRUE;
    END_IF
    IF EDGENEG(P1_Srobovanie.RR_ZapniHrniec_M4) THEN
        ZapniHrniec:= FALSE;
    END_IF

    //Zrušenie signálu skrutka pripravená//
    IF SkrutkovaciSet.SkrutkaPripravena=1 THEN
        IF SkrutkovaciSet.SkrutkaOdobrata=1 THEN
            SkrutkovaciSet.SkrutkaPripravena:=0;
        END_IF
    END_IF

    (********************Vreteno********************************)
    CASE SkrutkovaciSet.VretenoFaza OF
        0: SkrutkovaciSet.VretenoStatus:="Vypnute";
            SkrutkovaciSet.Vreteno.OUT.BlastAirBrake:=0;
            SkrutkovaciSet.Vreteno.OUT.BrakeSpindle:=0;
            SkrutkovaciSet.Vreteno.OUT.CounterBlast:=0;
            SkrutkovaciSet.Vreteno.OUT.Spindle:=0;
            SkrutkovaciSet.Vreteno.OUT.Vacuum:=0;
            SkrutkovaciSet.Vreteno.OUT.WasteExtraction:=0;

            SkrutkovaciSet.Zasobnik.OUT.Escapement:=0;
            SkrutkovaciSet.Zasobnik.OUT.FeedAir:=0;

            SkrutkovaciSet.Zasobnik.OUT.StartA20:=0;

            SkrutkovaciSet.CistenieVykonane:=0;
            SkrutkovaciSet.SkrutkaPripravena:=0;

            TprazdnyZasobnik.IN:=0;
            TakumulaciaPlna.IN:=0;
            TvytvorenieVakua.IN:=0;
            TodvetranieVakua.IN:=0;
            TprefukPredBrzdou.IN:=0;
            TprefukZaBrzdou.IN:=0;
            TvysuvanieSpindle.IN:=0;
            TpripravaSkrutky.IN:=0;
            ToddelovacZakladnaPoloha.IN:=0;
            TodsatieNecistot.IN:=0;
            TpodaniaSkrutky.IN:= 0;
            TpredSkrutkaPripravena.IN:= 0;
            TalarmuVysunutiaSkrutkovacky.IN:= 0;
            ZapniHrniec:= 0;
            PocetPokusovOpripravuSkrutky:=0;
            StavSkrutkovackaVysunuta:= 0;
            SkrutkovaciSet.VretenoFaza:=1;

        1: SkrutkovaciSet.VretenoStatus:="Inicializacia: cakam na povel";
            IF SkrutkovaciSet.Automat=1 THEN
                SkrutkovaciSet.CistenieVykonane:=0;
                SkrutkovaciSet.SkrutkaPripravena:=0;
                SkrutkovaciSet.VretenoFaza:=2;
            ELSIF SkrutkovaciSet.Manual=1 THEN
                SkrutkovaciSet.VretenoFaza:=250;
            END_IF

        2: SkrutkovaciSet.VretenoStatus:="Inicializacia: cakam na povel precisti hadice";

            IF SkrutkovaciSet.VykonajCistenie=1 THEN
                SkrutkovaciSet.Vreteno.OUT.Vacuum:=1;
                SkrutkovaciSet.VretenoFaza:=3;
            END_IF

        3: SkrutkovaciSet.VretenoStatus:="Inicializacia: Cakam na snimac: vreteno vysunute";
            SkrutkovaciSet.Vreteno.OUT.Spindle:=1;
            TalarmuVysunutiaSkrutkovacky.IN:= 1;

            IF P1_Srobovanie.IN.SkrutkM4_VysunutieHrotu_IOS10 > 1 THEN
                StavSkrutkovackaVysunuta:= TRUE;
                TvysuvanieSpindle.IN:=1;
            END_IF

            IF TvysuvanieSpindle.Q=1 AND StavSkrutkovackaVysunuta THEN
                TodvetranieVakua.IN:= 1;
                SkrutkovaciSet.Vreteno.OUT.CounterBlast:=1;
                SkrutkovaciSet.Vreteno.OUT.Vacuum:=0;
            END_IF

            IF TvysuvanieSpindle.Q AND StavSkrutkovackaVysunuta AND TodvetranieVakua.Q THEN
                StavSkrutkovackaVysunuta:= FALSE;
                TalarmuVysunutiaSkrutkovacky.IN:= 0;
                TvysuvanieSpindle.IN:=0;
                TodvetranieVakua.IN:= 0;
                SkrutkovaciSet.VretenoFaza:=4;
            ELSIF TalarmuVysunutiaSkrutkovacky.Q THEN
                P1_Alarmy[144]:= TRUE;
                P1_PoruchaST2:= TRUE;
            END_IF

        4: SkrutkovaciSet.VretenoStatus:="Inicializacia: Cakam na snimac: vreteno zasunute";
            SkrutkovaciSet.Vreteno.OUT.Spindle:=0;
            IF SkrutkovaciSet.Vreteno.IN.DeptControl=1 THEN
                SkrutkovaciSet.Vreteno.OUT.CounterBlast:=0;
                SkrutkovaciSet.VretenoFaza:=5;
            END_IF

        5: SkrutkovaciSet.VretenoStatus:="Inicializacia: Cakam na prefuknutie hadice za brzdou";
            TprefukZaBrzdou.IN:=1;
            SkrutkovaciSet.Vreteno.OUT.BlastAirBrake:=1;
            IF TprefukZaBrzdou.Q=1 THEN
                TprefukZaBrzdou.IN:=0;
                SkrutkovaciSet.Vreteno.OUT.BlastAirBrake:=0;
                SkrutkovaciSet.VretenoFaza:=6;
            END_IF

        6: SkrutkovaciSet.VretenoStatus:="Inicializacia: vypinam prefuk";
            TprefukZaBrzdou.IN:=0;
            SkrutkovaciSet.Vreteno.OUT.BlastAirBrake:=0;
            SkrutkovaciSet.Vreteno.OUT.Vacuum:=1;
            SkrutkovaciSet.VretenoFaza:=7;

        7: SkrutkovaciSet.VretenoStatus:="Inicializacia: Cakam na snimac: vreteno vysunute";
            SkrutkovaciSet.Vreteno.OUT.Spindle:=1;
            TalarmuVysunutiaSkrutkovacky.IN:= 1;

            IF P1_Srobovanie.IN.SkrutkM4_VysunutieHrotu_IOS10 > 1 THEN
                StavSkrutkovackaVysunuta:= TRUE;
                TvysuvanieSpindle.IN:=1;
            END_IF

            IF TvysuvanieSpindle.Q=1 AND StavSkrutkovackaVysunuta THEN
                TodvetranieVakua.IN:= 1;
                SkrutkovaciSet.Vreteno.OUT.CounterBlast:=1;
                SkrutkovaciSet.Vreteno.OUT.Vacuum:=0;
            END_IF

            IF TvysuvanieSpindle.Q AND StavSkrutkovackaVysunuta AND TodvetranieVakua.Q THEN
                StavSkrutkovackaVysunuta:= FALSE;
                TalarmuVysunutiaSkrutkovacky.IN:= 0;
                TvysuvanieSpindle.IN:=0;
                TodvetranieVakua.IN:= 0;
                SkrutkovaciSet.VretenoFaza:=8;
            ELSIF TalarmuVysunutiaSkrutkovacky.Q THEN
                P1_Alarmy[144]:= TRUE;
                P1_PoruchaST2:= TRUE;
            END_IF

        8: SkrutkovaciSet.VretenoStatus:="Inicializacia: Cakam na snimac: vreteno zasunute";
            SkrutkovaciSet.Vreteno.OUT.Spindle:=0;
            IF SkrutkovaciSet.Vreteno.IN.DeptControl=1 THEN
                SkrutkovaciSet.Vreteno.OUT.CounterBlast:=0;
                SkrutkovaciSet.VretenoFaza:=9;
            END_IF

        9: SkrutkovaciSet.VretenoStatus:="Inicializacia: Cakam na prefuknutie hadice pred brzdou";
            TprefukPredBrzdou.IN:=1;
            SkrutkovaciSet.Zasobnik.OUT.FeedAir:=1;
            IF TprefukPredBrzdou.Q=1 THEN
                TprefukPredBrzdou.IN:=0;
                SkrutkovaciSet.Zasobnik.OUT.FeedAir:=0;
                SkrutkovaciSet.VretenoFaza:=10;
            END_IF

        10: SkrutkovaciSet.VretenoStatus:="Inicializacia: Cakam na snimac: brzda uvolnena";
            SkrutkovaciSet.Vreteno.OUT.BrakeSpindle:=1;
            IF SkrutkovaciSet.Vreteno.IN.BrakeOpen=1 THEN
                SkrutkovaciSet.Vreteno.OUT.BlastAirBrake:=1;
                SkrutkovaciSet.VretenoFaza:=11;
            END_IF

        11: SkrutkovaciSet.VretenoStatus:="Inicializacia: Cakam na prefuknutie hadice za brzdou";
            TprefukZaBrzdou.IN:=1;
            SkrutkovaciSet.Vreteno.OUT.BlastAirBrake:=1;
            IF TprefukZaBrzdou.Q=1 THEN
                TprefukZaBrzdou.IN:=0;
                SkrutkovaciSet.Vreteno.OUT.BlastAirBrake:=0;
                SkrutkovaciSet.VretenoFaza:=12;
            END_IF

        12: SkrutkovaciSet.VretenoStatus:="Inicializacia: vypinam prefuk";
            TprefukZaBrzdou.IN:=0;
            SkrutkovaciSet.Vreteno.OUT.BlastAirBrake:=0;
            SkrutkovaciSet.Vreteno.OUT.Vacuum:=1;
            SkrutkovaciSet.VretenoFaza:=13;

        13: SkrutkovaciSet.VretenoStatus:="Inicializacia: Cakam na snimac: vreteno vysunute";
            SkrutkovaciSet.Vreteno.OUT.Spindle:=1;
            TalarmuVysunutiaSkrutkovacky.IN:= 1;

            IF P1_Srobovanie.IN.SkrutkM4_VysunutieHrotu_IOS10 > 1 THEN
                StavSkrutkovackaVysunuta:= TRUE;
                TvysuvanieSpindle.IN:=1;
            END_IF

            IF TvysuvanieSpindle.Q=1 AND StavSkrutkovackaVysunuta THEN
                TodvetranieVakua.IN:= 1;
                SkrutkovaciSet.Vreteno.OUT.CounterBlast:=1;
                SkrutkovaciSet.Vreteno.OUT.Vacuum:=0;
            END_IF

            IF TvysuvanieSpindle.Q AND StavSkrutkovackaVysunuta AND TodvetranieVakua.Q THEN
                StavSkrutkovackaVysunuta:= FALSE;
                TalarmuVysunutiaSkrutkovacky.IN:= 0;
                TvysuvanieSpindle.IN:=0;
                TodvetranieVakua.IN:= 0;
                SkrutkovaciSet.VretenoFaza:=14;
            ELSIF TalarmuVysunutiaSkrutkovacky.Q THEN
                P1_Alarmy[144]:= TRUE;
                P1_PoruchaST2:= TRUE;
            END_IF

        14: SkrutkovaciSet.VretenoStatus:="Inicializacia: Cakam na snimac: vreteno zasunute";
            SkrutkovaciSet.Vreteno.OUT.Spindle:=0;
            IF SkrutkovaciSet.Vreteno.IN.DeptControl=1 THEN
                SkrutkovaciSet.Vreteno.OUT.CounterBlast:=0;
                SkrutkovaciSet.VretenoFaza:=15;
            END_IF

        15: SkrutkovaciSet.VretenoStatus:="Inicializacia: Cakam na snimac: brzda zasunuta";
            SkrutkovaciSet.Vreteno.OUT.BrakeSpindle:=0;
            IF SkrutkovaciSet.Vreteno.IN.BrakeClosed=1 THEN
                SkrutkovaciSet.CistenieVykonane:=1;
                SkrutkovaciSet.VretenoFaza:=16;
            END_IF

        16: SkrutkovaciSet.VretenoStatus:="Inicializacia: Cakam na zrusenie signalu: vykonaj cistenie";
            IF SkrutkovaciSet.VykonajCistenie=0 THEN
                SkrutkovaciSet.CistenieVykonane:=0;
                SkrutkovaciSet.SkrutkaPripravena:=0;
                SkrutkovaciSet.VretenoFaza:=100;
            END_IF

        100: SkrutkovaciSet.VretenoStatus:="Cakam kym zasobnik pripravy skrutku";
            ZapniHrniec:= 1;
            IF TakumulaciaPlna.Q=1 AND SkrutkovaciSet.Zasobnik.OUT.StartA20 THEN
                TpodaniaSkrutky.IN:= 1;
            END_IF

            IF TpodaniaSkrutky.Q THEN
                TpodaniaSkrutky.IN:= 0;
                SkrutkovaciSet.VretenoFaza:=102;
            END_IF

        102: SkrutkovaciSet.VretenoStatus:="Cakam na snimac: skrutka presla hadicou";
            SkrutkovaciSet.Zasobnik.OUT.Escapement:=1;
            TpripravaSkrutky.IN:=1;
            IF SkrutkovaciSet.Zasobnik.IN.ScrewMeasurement=1 THEN
                SkrutkovaciSet.Zasobnik.OUT.FeedAir:=1;
                TpripravaSkrutky.IN:=0;
                SkrutkovaciSet.VretenoFaza:=104;
            ELSIF TpripravaSkrutky.Q=1 THEN
                TpripravaSkrutky.IN:=0;
                SkrutkovaciSet.Zasobnik.OUT.Escapement:=0;
                SkrutkovaciSet.VretenoFaza:=100;
            END_IF

        104: SkrutkovaciSet.VretenoStatus:="Cakam na snimac: skrutka presla hadicou pred brzdou";
            IF SkrutkovaciSet.Vreteno.IN.ScrewMeasurementBrake=1 THEN
                SkrutkovaciSet.Zasobnik.OUT.Escapement:=0;
                SkrutkovaciSet.Zasobnik.OUT.FeedAir:=0;
                PocetPokusovOpripravuSkrutky:=0;
                SkrutkovaciSet.VretenoFaza:=106;
            END_IF

        106: SkrutkovaciSet.VretenoStatus:="Cakam na odsatie necistot";
            SkrutkovaciSet.Vreteno.OUT.WasteExtraction:=1;
            TodsatieNecistot.IN:=1;

            IF TodsatieNecistot.Q=1 THEN
                TodsatieNecistot.IN:=0;
                SkrutkovaciSet.Vreteno.OUT.WasteExtraction:=0;
                SkrutkovaciSet.VretenoFaza:=107;
            END_IF

        107: SkrutkovaciSet.VretenoStatus:="Cakam kym skrutkovacka odoberie skrutku";
            IF SkrutkovaciSet.SkrutkaPripravena=0 AND SkrutkovaciSet.SkrutkaOdobrata=0 THEN
                SkrutkovaciSet.VretenoFaza:=108;
            END_IF

        108: SkrutkovaciSet.VretenoStatus:="Cakam na snimac: brzda uvolnena";
            SkrutkovaciSet.Vreteno.OUT.BrakeSpindle:=1;
            IF SkrutkovaciSet.Vreteno.IN.BrakeOpen=1 THEN
                SkrutkovaciSet.Vreteno.OUT.BlastAirBrake:=1;
                SkrutkovaciSet.VretenoFaza:=110;
            END_IF

        110: SkrutkovaciSet.VretenoStatus:="Cakam na snimac: skrutka presla hadicou pred vretenom";
            IF SkrutkovaciSet.Vreteno.IN.ScrewMeasurement=1 THEN
                SkrutkovaciSet.Vreteno.OUT.BlastAirBrake:=0;
                SkrutkovaciSet.Vreteno.OUT.BrakeSpindle:=0;
                SkrutkovaciSet.VretenoFaza:=112;
            END_IF

        112: SkrutkovaciSet.VretenoStatus:="Cakam na snimac: brzda zabrzdena";
            SkrutkovaciSet.Vreteno.OUT.BrakeSpindle:=0;
            IF SkrutkovaciSet.Vreteno.IN.BrakeClosed=1 AND SkrutkovaciSet.SkrutkaOdobrata=0 THEN
                TpredSkrutkaPripravena.IN:= 1;
                IF TpredSkrutkaPripravena.Q THEN
                    TpredSkrutkaPripravena.IN:= 0;
                    SkrutkovaciSet.SkrutkaPripravena:=1;
                    SkrutkovaciSet.VretenoFaza:=100;
                END_IF
            END_IF

            //*************** opakovany pokus o oddelenie skrutky *********************************

        170: SkrutkovaciSet.VretenoStatus:="Cakam na presunutie oddelovaca do zakladnej polohy";
            SkrutkovaciSet.Zasobnik.OUT.Escapement:=0;
            ToddelovacZakladnaPoloha.IN:=1;
            IF ToddelovacZakladnaPoloha.Q=1 THEN
                ToddelovacZakladnaPoloha.IN:=0;
                PocetPokusovOpripravuSkrutky:=PocetPokusovOpripravuSkrutky+1;
                IF PocetPokusovOpripravuSkrutky>3 THEN
                    PocetPokusovOpripravuSkrutky:=0;
                    SkrutkovaciSet.VretenoFaza:=171;
                ELSE
                    SkrutkovaciSet.VretenoFaza:=100;
                END_IF
            END_IF

        171: SkrutkovaciSet.VretenoStatus:="Zaseknuta skrutka v oddelovaci!!!";
    END_CASE

END_PROGRAM

PROGRAM _EXIT
	(* Insert code here *)

END_PROGRAM
```

#### Types.typ - Local data types
```iecst
TYPE
	SkrutkovaciSetStruc : 	STRUCT
		VretenoStatus : WSTRING[80];
		VretenoFaza : USINT;
		Zasobnik : ZasobnikStruc;
		Vreteno : VretenoStruc;
		SkrutkaOdobrata : BOOL;
		SkrutkaPripravena : BOOL;
		Manual : BOOL;
		PodajSrobu : BOOL;
		CistenieVykonane : BOOL;
		VykonajCistenie : BOOL;
		Automat : BOOL;
	END_STRUCT;
	INzasobnik : 	STRUCT
		AccumulationSwitch : BOOL; (*Snimac zaplnenia S25*)
		ScrewMeasurement : BOOL; (*Kontrola matice S21*)
		FeederLevelControl : BOOL; (*Hladina v zasobniku S20*)
	END_STRUCT;
	OUTzasobnik : 	STRUCT
		StartA20 : BOOL; (*Zapnutie vibrovania A20*)
		Escapement : BOOL; (*Pustanie matky do hadice Y22*)
		FeedAir : BOOL; (*Strielanie do hadice Y21*)
		SortingAir : BOOL; (*Triedenie kusov Y30*)
		BlowOff : BOOL; (*Zhadzovanie kusov Y25*)
	END_STRUCT;
	INvreteno : 	STRUCT
		ReturnStroke : BOOL; (*Vreteno zasunute S01*)
		DeptControl : BOOL; (*Vreteno vysunute S02*)
		BrakeClosed : BOOL; (*Brzda zatvorena S13*)
		BrakeOpen : BOOL; (*Brzda otvorena S12*)
		ScrewMeasurementBrake : BOOL; (*Kontrola matice pred brzdou S15*)
		ScrewMeasurement : BOOL; (*Kontrola matice v hadici S06*)
	END_STRUCT;
	OUTvreteno : 	STRUCT
		WasteExtraction : BOOL; (*Odstranovanie spiny Y13*)
		Spindle : BOOL; (*Vysunutie vretena Y02*)
		BlastAirBrake : BOOL; (*Strielanie za brzdou Y14*)
		BrakeSpindle : BOOL; (*Brzda vretena Y12*)
		Vacuum : BOOL; (*Pridrzanie skrutky Y15*)
		CounterBlast : BOOL; (*Uvolnenie skrutky Y16*)
	END_STRUCT;
	VretenoStruc : 	STRUCT
		OUT : OUTvreteno;
		IN : INvreteno;
	END_STRUCT;
	ZasobnikStruc : 	STRUCT
		OUT : OUTzasobnik;
		IN : INzasobnik;
	END_STRUCT;
END_TYPE
```

#### Variables.var - Local variables
```iecst
VAR
	SkrutkovaciSet : SkrutkovaciSetStruc;
	TprazdnyZasobnik : TON;
	TakumulaciaPlna : TON;
	TvytvorenieVakua : TON;
	TodvetranieVakua : TON;
	TprefukPredBrzdou : TON;
	TvysuvanieSpindle : TON;
	TprefukZaBrzdou : TON;
	PocetPokusovOpripravuSkrutky : USINT;
	ToddelovacZakladnaPoloha : TON;
	TpripravaSkrutky : TON;
	TodsatieNecistot : TON;
	Tvibrovanie : TON;
	TvyfukovaniePredVibrovanim : TON;
	ZapniHrniec : BOOL;
	TpodaniaSkrutky : TON;
	TpredSkrutkaPripravena : TON;
	TvypnutieOfuku : TON;
	StavSkrutkovackaVysunuta : BOOL;
	TalarmuVysunutiaSkrutkovacky : TON;
END_VAR
```

### Program Logical/Program/Pracovisko_1/P1_AkumulacnyStoper (IEC)

#### Main.st - Init, cyclic, exit code
```iecst
PROGRAM _INIT
	(* Insert code here *)

END_PROGRAM

PROGRAM _CYCLIC

	//Volanie funkcie SequenceControl//
	SequenceControl(SC:= SC_P1_AkumulacnyStoper);

	//Reset sekcie //
	IF NOT Safety.STAV.P1_ZonaBunky_AKTIVNA THEN
		SC_P1_AkumulacnyStoper.Step:= 0;
	ELSIF P1_AkumulacnyStoper.Reset THEN
		SC_P1_AkumulacnyStoper.Step:= 0;
		P1_AkumulacnyStoper.Reset:= FALSE;
	END_IF

	CASE SC_P1_AkumulacnyStoper.Step OF

		0:
			SC_P1_AkumulacnyStoper.StepName:='0 - Nulovanie';
			P1_AkumulacnyStoper.Automat:= FALSE;
			P1_AkumulacnyStoper.KoniecCyklu:= FALSE;
			P1_AkumulacnyStoper.Manual:= FALSE;
			P1_AkumulacnyStoper.STAV.PoINIT:= FALSE;
			P1_AkumulacnyStoper.OUT.ZasunStoper_YV74:= FALSE;

			IF Safety.STAV.P1_ZonaBunky_AKTIVNA AND NOT P1_Pracovisko.STAV.PORUCHA AND P1_Pracovisko.IN.PrivodVzduchu_SnimacTlaku_S18 THEN
				SC_P1_AkumulacnyStoper.ResetStep:= TRUE;
				SC_P1_AkumulacnyStoper.Step:= 1;
			END_IF

		1:
			SC_P1_AkumulacnyStoper.StepName:='1 - Cakam na spustenie vyroby';
			P1_AkumulacnyStoper.KoniecCyklu:= FALSE;
            IF P1_AkumulacnyStoper.Automat THEN
				SC_P1_AkumulacnyStoper.Step:= 2;
			ELSIF P1_AkumulacnyStoper.Manual THEN
				SC_P1_AkumulacnyStoper.Step:= 700;
			END_IF

			//********************************************************Inicializácia****************************************************************************//
		2:
			SC_P1_AkumulacnyStoper.StepName:='2 - Inicializacia - cakam na spustenie inicializacie';
			SC_P1_AkumulacnyStoper.IdleTime.PT:= T#4s;
			SC_P1_AkumulacnyStoper.AlarmTime.PT:= T#5s;

			IF P1_Dopravniky.STAV.PoINIT THEN
				SC_P1_AkumulacnyStoper.ResetStep:= TRUE;
				SC_P1_AkumulacnyStoper.Step:= 3;
			END_IF

		3:
			SC_P1_AkumulacnyStoper.StepName:='3 - Inicializacia - hladanie paletky';
			SC_P1_AkumulacnyStoper.IdleTime.PT:= T#5s;
			SC_P1_AkumulacnyStoper.AlarmTime.PT:= T#5s;
			SC_P1_AkumulacnyStoper.IdleTime.IN:= TRUE;

			IF P1_AkumulacnyStoper.IN.PritomnPaletky_IS45 THEN
				P1_AkumulacnyStoper.STAV.PoINIT:= TRUE;
				SC_P1_AkumulacnyStoper.ResetStep:= TRUE;
				SC_P1_AkumulacnyStoper.Step:= 101;
			ELSIF SC_P1_AkumulacnyStoper.IdleTime.Q THEN
				P1_AkumulacnyStoper.STAV.PoINIT:= TRUE;
				SC_P1_AkumulacnyStoper.ResetStep:= TRUE;
				SC_P1_AkumulacnyStoper.Step:= 100;
			END_IF

			//********************************************************Automatický režim****************************************************************************//
		100:
			SC_P1_AkumulacnyStoper.StepName:='100 - Automaticky Rezim - cakam na príchod paletky na stoper';
			SC_P1_AkumulacnyStoper.IdleTime.PT:= T#200ms;
			SC_P1_AkumulacnyStoper.AlarmTime.PT:= T#5s;

            SC_P1_AkumulacnyStoper.IdleTime.IN:= P1_AkumulacnyStoper.IN.PritomnPaletky_IS45;

            IF P1_AkumulacnyStoper.KoniecCyklu THEN
                SC_P1_AkumulacnyStoper.ResetStep:= TRUE;
                SC_P1_AkumulacnyStoper.Step:= 0;
            ELSIF SC_P1_AkumulacnyStoper.IdleTime.Q THEN
				P1_StoperSrobovania.STAV.PrebiehaVyvezeniePaletky:= FALSE;
                SC_P1_AkumulacnyStoper.ResetStep:= TRUE;
				SC_P1_AkumulacnyStoper.Step:= 101;
			END_IF

		101:
			SC_P1_AkumulacnyStoper.StepName:='101 - Automaticky Rezim - cakam na vyvezenie paletky na stoper zakladania tesnenia';
			SC_P1_AkumulacnyStoper.IdleTime.PT:= T#200ms;
			SC_P1_AkumulacnyStoper.AlarmTime.PT:= T#5s;

            IF P1_AkumulacnyStoper.KoniecCyklu THEN
                SC_P1_AkumulacnyStoper.ResetStep:= TRUE;
                SC_P1_AkumulacnyStoper.Step:= 0;
            ELSIF SC_P2_StoperZaklTesnenia.Step = 100 AND NOT P2_StoperZaklTesnenia.IN.PritomnostPaletky_S6 AND Safety.STAV.P2_ZaklTesnenia_Pojazd_ZASUNUTY THEN
				SC_P1_AkumulacnyStoper.ResetStep:= TRUE;
				SC_P1_AkumulacnyStoper.Step:= 105;
			ELSIF NOT P1_AkumulacnyStoper.IN.PritomnPaletky_IS45 THEN
				SC_P1_AkumulacnyStoper.ResetStep:= TRUE;
				SC_P1_AkumulacnyStoper.Step:= 100;
			END_IF

		105:
			SC_P1_AkumulacnyStoper.StepName:='105 - Automaticky Rezim - vyvazam paletku na stoper zakladania tesnenia';
			SC_P1_AkumulacnyStoper.IdleTime.PT:= T#200ms;
			SC_P1_AkumulacnyStoper.AlarmTime.PT:= T#10s;

			IF NOT SC_P1_AkumulacnyStoper.Switch1 THEN
				P1_AkumulacnyStoper.OUT.ZasunStoper_YV74:= TRUE;
				SC_P1_AkumulacnyStoper.AlarmTime.IN:= TRUE;
                SC_P1_AkumulacnyStoper.Switch1:= TRUE;
			END_IF

			IF NOT P1_AkumulacnyStoper.IN.PritomnPaletky_IS45 THEN
                P1_AkumulacnyStoper.OUT.ZasunStoper_YV74:= FALSE;
                SC_P1_AkumulacnyStoper.AlarmTime.IN:= FALSE;
			END_IF

			IF P2_StoperZaklTesnenia.IN.PritomnostPaletky_S6 THEN
				SC_P1_AkumulacnyStoper.ResetStep:= TRUE;
                SC_P1_AkumulacnyStoper.Step:= 100;
            ELSIF  SC_P1_AkumulacnyStoper.AlarmTime.Q THEN
                P1_Alarmy[162]:= TRUE;
                P1_Pracovisko.KoniecCyklu:= TRUE;
                SC_P1_AkumulacnyStoper.ResetStep:= TRUE;
                SC_P1_AkumulacnyStoper.Step:= 0;
			END_IF

			//*******************************************************Manuálny režim*******************************************************************************//
		700:
			SC_P1_AkumulacnyStoper.StepName:='700 - Manualny Rezim';
			SC_P1_AkumulacnyStoper.IdleTime.PT:= T#8s;
			SC_P1_AkumulacnyStoper.AlarmTime.PT:= T#5s;

	END_CASE

END_PROGRAM

PROGRAM _EXIT
	(* Insert code here *)

END_PROGRAM
```

### Program Logical/Program/Pracovisko_1/P1_Robot (IEC)

#### Main.st - Init, cyclic, exit code
```iecst
PROGRAM _INIT
    Triger_0:= FALSE;

END_PROGRAM

PROGRAM _CYCLIC

	//Volanie funkcie SequenceControl//
    SequenceControl(SC:= SC_P1_Robot);

    //Volanie podprogramov//
    IOLinkKomunikacia;
    ProfinetKomunikaciaRobot;

    //Reset sekcie //
    IF NOT Safety.STAV.ZonaCS_AKTIVNA THEN
        SC_P1_Robot.Step:= 0;
    ELSIF P1_PoruchaST2 THEN
        SC_P1_Robot.Step:= 0;
    ELSIF P1_Robot.Reset THEN
        SC_P1_Robot.Step:= 0;
        P1_Robot.Reset:= FALSE;
    END_IF

    IF NOT Safety.STAV.P1_ZonaBunky_AKTIVNA AND NOT Triger_0 THEN
        Triger_0:= TRUE;
        SC_P1_Robot.Step:= 0;
    END_IF

    IF Safety.STAV.P1_ZonaBunky_AKTIVNA THEN
        Triger_0:= FALSE;
    END_IF

    CASE SC_P1_Robot.Step OF

        0:
            SC_P1_Robot.StepName:='0 - Nulovanie';
            P1_Robot.Automat:= FALSE;
            P1_Robot.KoniecCyklu:= FALSE;
            P1_Robot.Manual:= FALSE;
            P1_Robot.Reset:= FALSE;
            P1_Robot.STAV.PoINIT:= FALSE;
            P1_Robot.KOM_OUT.Odparkovanie:= FALSE;
            P1_Robot.KOM_OUT.PP_na_Main:= FALSE;
            P1_Robot.KOM_OUT.Reset_CS:= FALSE;
            P1_Robot.KOM_OUT.StartProgramu:= FALSE;
            P1_Robot.KOM_OUT.StartProgramuMain:= FALSE;
            P1_Robot.KOM_OUT.VypniMotory:= FALSE;
            P1_Robot.KOM_OUT.ZapniMotory:= FALSE;
            IF P1_Robot.KOM_IN.Stav_RezimAUTOMAT AND P1_Robot.KOM_IN.Stav_ProgramRUN THEN
                P1_Robot.KOM_OUT.StopProgramu:= TRUE;
            ELSE
                P1_Robot.KOM_OUT.StopProgramu:= FALSE;
            END_IF
            IF Safety.STAV.ZonaCS_AKTIVNA AND Safety.STAV.P1_ZonaBunky_AKTIVNA AND NOT P1_Pracovisko.STAV.PORUCHA AND P1_Pracovisko.IN.PrivodVzduchu_SnimacTlaku_S18 AND NOT P1_Robot.KOM_IN.Stav_ProgramRUN THEN
                P1_Robot.KOM_OUT.StopProgramu:= FALSE;
                SC_P1_Robot.ResetStep:= TRUE;
                SC_P1_Robot.Step:= 1;
            END_IF

        1:
            SC_P1_Robot.StepName:='1 - Cakam na spustenie vyroby';
            P1_Robot.KoniecCyklu:= FALSE;
            IF P1_Robot.Automat THEN
                SC_P1_Robot.Step:= 2;
            ELSIF P1_Robot.Manual THEN
                SC_P1_Robot.Step:= 700;
            END_IF

            //********************************************************Inicializácia****************************************************************************//

        2:
            SC_P1_Robot.StepName:='2 - Inicializacia - cakam na spustenie inicializacie';
            SC_P1_Robot.IdleTime.PT:= T#500ms;
            SC_P1_Robot.AlarmTime.PT:= T#5s;

            SC_P1_Robot.IdleTime.IN:= TRUE;

            IF SC_P1_Robot.IdleTime.Q THEN
                SC_P1_Robot.ResetStep:= TRUE;
                SC_P1_Robot.Step:= 3;
            END_IF

        3:
            SC_P1_Robot.StepName:='2 - Inicializacia - kontrolujem central stop robota';
            SC_P1_Robot.IdleTime.PT:= T#500ms;
            SC_P1_Robot.AlarmTime.PT:= T#5s;

            IF P1_Robot.KOM_IN.Stav_RobotCS THEN
                P1_Robot.KOM_OUT.Reset_CS:= TRUE;
            END_IF

            IF NOT P1_Robot.KOM_IN.Stav_RobotCS THEN
                P1_Robot.KOM_OUT.Reset_CS:= FALSE;
                SC_P1_Robot.ResetStep:= TRUE;
                SC_P1_Robot.Step:= 4;
            END_IF

        4:
            SC_P1_Robot.StepName:='4 - Inicializacia - zapinam motory robota';
            SC_P1_Robot.IdleTime.PT:= T#500ms;
            SC_P1_Robot.AlarmTime.PT:= T#5s;

            IF NOT P1_Robot.KOM_IN.Stav_MotoryON THEN
                P1_Robot.KOM_OUT.ZapniMotory:= TRUE;
            END_IF

            IF P1_Robot.KOM_IN.Stav_MotoryON THEN
                P1_Robot.KOM_OUT.ZapniMotory:= FALSE;
                SC_P1_Robot.ResetStep:= TRUE;
                SC_P1_Robot.Step:= 6;
            END_IF

        6:
            SC_P1_Robot.StepName:='6 - Inicializacia - spustam program robota od zaciatku';
            SC_P1_Robot.IdleTime.PT:= T#500ms;
            SC_P1_Robot.AlarmTime.PT:= T#5s;

            IF NOT SC_P1_Robot.Switch1 THEN
                P1_Robot.KOM_OUT.StartProgramuMain:= TRUE;
                SC_P1_Robot.Switch1:= TRUE;
            END_IF

            IF P1_Robot.KOM_IN.Stav_ProgramRUN AND P1_Robot.KOM_IN.Stav_VystupyZresetovane THEN
                P1_Robot.KOM_OUT.StartProgramuMain:= FALSE;
                P1_Robot.STAV.PoINIT:= TRUE;
                SC_P1_Robot.ResetStep:= TRUE;
                SC_P1_Robot.Step:= 100;
            END_IF

            //********************************************************Automatický režim****************************************************************************//

        100:
            SC_P1_Robot.StepName:='100 - Automaticky Rezim - cakam na ukoncenie programu robota';
            SC_P1_Robot.IdleTime.PT:= T#200ms;
            SC_P1_Robot.AlarmTime.PT:= T#5s;

            IF P1_Robot.KoniecCyklu AND NOT P1_StoperSrobovania.Automat THEN
                SC_P1_Robot.ResetStep:= TRUE;
                SC_P1_Robot.Step:= 0;
            END_IF

            //*******************************************************Manuálny režim*******************************************************************************//

        700:
            SC_P1_Robot.StepName:='700 - Manualny Rezim';
            SC_P1_Robot.IdleTime.PT:= T#8s;
            SC_P1_Robot.AlarmTime.PT:= T#5s;

    END_CASE

END_PROGRAM

PROGRAM _EXIT
	(* Insert code here *)

END_PROGRAM
```

#### Variables.var - Local variables
```iecst
VAR
	Triger_0 : BOOL;
END_VAR
```

#### IOLinkKomunikacia.st
```iecst
ACTION IOLinkKomunikacia:

	//Modul ovládania gripra//
	P1_Robot.IN.Griper_Otvoreny_MS40:=	P1_Robot.PAR.Modul_IOLink_Inputs.0;
	P1_Robot.IN.Griper_Zatvoreny_MS41:=	P1_Robot.PAR.Modul_IOLink_Inputs.1;
	P1_Robot.PAR.Modul_IOLink_Inputs.2;
	P1_Robot.PAR.Modul_IOLink_Inputs.3;
	P1_Robot.PAR.Modul_IOLink_Inputs.4;
	P1_Robot.PAR.Modul_IOLink_Inputs.5;
	P1_Robot.IN.KodGripra_Bit0:= P1_Robot.PAR.Modul_IOLink_Inputs.6;
	P1_Robot.IN.KodGripra_Bit1:= P1_Robot.PAR.Modul_IOLink_Inputs.7;

	//Typ gripra//
	IF P1_Robot.IN.KodGripra_Bit0 AND NOT P1_Robot.IN.KodGripra_Bit1 THEN
		P1_Robot.KOM_OUT.TypGripra_5H:= FALSE;
		P1_Robot.KOM_OUT.TypGripra_45F:= TRUE;
	ELSIF NOT P1_Robot.IN.KodGripra_Bit0 AND P1_Robot.IN.KodGripra_Bit1 THEN
		P1_Robot.KOM_OUT.TypGripra_45F:= FALSE;
		P1_Robot.KOM_OUT.TypGripra_5H:= TRUE;
	ELSE
		P1_Robot.KOM_OUT.TypGripra_45F:= FALSE;
		P1_Robot.KOM_OUT.TypGripra_5H:= FALSE;
	END_IF

END_ACTION
```

#### ProfinetKomunikaciaRobot.st
```iecst
ACTION ProfinetKomunikaciaRobot:

	//Vstupy z Robota do PLC//
	P1_Robot.KOM_IN.Stav_RezimAUTOMAT:= P1_Robot.KOM_IN.Profinet_PLC_INPUTS[0].0;
	P1_Robot.KOM_IN.Stav_ProgramRUN:= P1_Robot.KOM_IN.Profinet_PLC_INPUTS[0].1;
	P1_Robot.KOM_IN.Stav_MotoryOFF:= P1_Robot.KOM_IN.Profinet_PLC_INPUTS[0].2;
	P1_Robot.KOM_IN.Stav_MotoryON:= P1_Robot.KOM_IN.Profinet_PLC_INPUTS[0].3;
	P1_Robot.KOM_IN.Stav_RobotCS:= P1_Robot.KOM_IN.Profinet_PLC_INPUTS[0].4;

	P1_Robot.KOM_IN.Stav_DPS_4F_Odobraty:= P1_Robot.KOM_IN.Profinet_PLC_INPUTS[1].0;
	P1_Robot.KOM_IN.Stav_DPS_4F_Polozeny:= P1_Robot.KOM_IN.Profinet_PLC_INPUTS[1].1;
	P1_Robot.KOM_IN.Stav_DPS_5F_Odobraty:= P1_Robot.KOM_IN.Profinet_PLC_INPUTS[1].2;
	P1_Robot.KOM_IN.Stav_DPS_5F_Polozeny:= P1_Robot.KOM_IN.Profinet_PLC_INPUTS[1].3;
	P1_Robot.KOM_IN.Stav_Foam4F_Odobraty:= P1_Robot.KOM_IN.Profinet_PLC_INPUTS[1].4;
	P1_Robot.KOM_IN.Stav_Foam4F_Polozeny:= P1_Robot.KOM_IN.Profinet_PLC_INPUTS[1].5;
	P1_Robot.KOM_IN.Stav_Foam5F_Odobraty:= P1_Robot.KOM_IN.Profinet_PLC_INPUTS[1].6;
	P1_Robot.KOM_IN.Stav_Foam5F_Polozeny:= P1_Robot.KOM_IN.Profinet_PLC_INPUTS[1].7;

	P1_Robot.KOM_IN.Stav_RobotBezpPozicia_Srobovanie:= P1_Robot.KOM_IN.Profinet_PLC_INPUTS[2].0;
	P1_Robot.KOM_IN.Stav_RobotOdparkovany:= P1_Robot.KOM_IN.Profinet_PLC_INPUTS[2].1;
	P1_Robot.KOM_IN.Stav_RobotPoziciaCakania:= P1_Robot.KOM_IN.Profinet_PLC_INPUTS[2].2;
	P1_Robot.KOM_IN.Stav_SpodnyBusbar4F_Odobraty:= P1_Robot.KOM_IN.Profinet_PLC_INPUTS[2].3;
	P1_Robot.KOM_IN.Stav_SpodnyBusbar4F_Polozeny:= P1_Robot.KOM_IN.Profinet_PLC_INPUTS[2].4;
	P1_Robot.KOM_IN.Stav_SpodnyBusbar5F_Odobraty:= P1_Robot.KOM_IN.Profinet_PLC_INPUTS[2].5;
	P1_Robot.KOM_IN.Stav_SpodnyBusbar5F_Polozeny:= P1_Robot.KOM_IN.Profinet_PLC_INPUTS[2].6;
	P1_Robot.KOM_IN.Stav_SpodnyBusbar5H_Odobraty:= P1_Robot.KOM_IN.Profinet_PLC_INPUTS[2].7;

	P1_Robot.KOM_IN.Stav_SpodnyBusbar5H_Polozeny:= P1_Robot.KOM_IN.Profinet_PLC_INPUTS[3].0;
    P1_Robot.KOM_IN.Stav_VystupyZresetovane:= P1_Robot.KOM_IN.Profinet_PLC_INPUTS[3].1;
    P1_Robot.KOM_IN.Stav_BusbaryUvolnene:= P1_Robot.KOM_IN.Profinet_PLC_INPUTS[3].2;
    P1_Robot.KOM_IN.Stav_RobotOdoberaBusbary:= P1_Robot.KOM_IN.Profinet_PLC_INPUTS[3].3;
    P1_Robot.KOM_IN.Stav_RobotOdoberaFoamy:= P1_Robot.KOM_IN.Profinet_PLC_INPUTS[3].4;

	P1_Robot.OUT.OdistiGriper_YV107:= P1_Robot.KOM_IN.Profinet_PLC_INPUTS[4].0;
	P1_Robot.OUT.ZaistiGriper_YV106:= P1_Robot.KOM_IN.Profinet_PLC_INPUTS[4].1;
	P1_Robot.OUT.OtvorGriper_YV97:= P1_Robot.KOM_IN.Profinet_PLC_INPUTS[4].2;
	P1_Robot.OUT.ZatvorGriper_YV98:= P1_Robot.KOM_IN.Profinet_PLC_INPUTS[4].3;
	P1_Robot.OUT.ZapniVakum_YV108:= P1_Robot.KOM_IN.Profinet_PLC_INPUTS[4].4;
	P1_Robot.OUT.VypniVakum_YV114:= P1_Robot.KOM_IN.Profinet_PLC_INPUTS[4].5;

	//Vystupy z PLC do Robota//
	P1_Robot.KOM_OUT.Profinet_PLC_OUTPUTS[0].0:= P1_Robot.KOM_OUT.VypniMotory;
	P1_Robot.KOM_OUT.Profinet_PLC_OUTPUTS[0].1:= P1_Robot.KOM_OUT.ZapniMotory;
	P1_Robot.KOM_OUT.Profinet_PLC_OUTPUTS[0].2:= P1_Robot.KOM_OUT.PP_na_Main;
	P1_Robot.KOM_OUT.Profinet_PLC_OUTPUTS[0].3:= P1_Robot.KOM_OUT.StartProgramu;
	P1_Robot.KOM_OUT.Profinet_PLC_OUTPUTS[0].4:= P1_Robot.KOM_OUT.StartProgramuMain;
	P1_Robot.KOM_OUT.Profinet_PLC_OUTPUTS[0].5:= P1_Robot.KOM_OUT.StopProgramu;
	P1_Robot.KOM_OUT.Profinet_PLC_OUTPUTS[0].6:= P1_Robot.KOM_OUT.Reset_CS;

	P1_Robot.KOM_OUT.Profinet_PLC_OUTPUTS[1].0:= P1_Robot.KOM_OUT.ManipSrobovania_BezpecnaPozicia;
	P1_Robot.KOM_OUT.Profinet_PLC_OUTPUTS[1].1:= P1_Robot.KOM_OUT.OdoberDPS_4F_z_Paletky;
	P1_Robot.KOM_OUT.Profinet_PLC_OUTPUTS[1].2:= P1_Robot.KOM_OUT.OdoberDPS_5F_z_Paletky;
	P1_Robot.KOM_OUT.Profinet_PLC_OUTPUTS[1].3:= P1_Robot.KOM_OUT.OdoberFoam4F_z_Paletky;
	P1_Robot.KOM_OUT.Profinet_PLC_OUTPUTS[1].4:= P1_Robot.KOM_OUT.OdoberFoam5F_z_Paletky;
	P1_Robot.KOM_OUT.Profinet_PLC_OUTPUTS[1].5:= P1_Robot.KOM_OUT.OdoberSpodnyBusbar4F_z_Paletky;
	P1_Robot.KOM_OUT.Profinet_PLC_OUTPUTS[1].6:= P1_Robot.KOM_OUT.OdoberSpodnyBusbar5F_z_Paletky;
	P1_Robot.KOM_OUT.Profinet_PLC_OUTPUTS[1].7:= P1_Robot.KOM_OUT.OdoberSpodnyBusbar5H_z_Paletky;

	P1_Robot.KOM_OUT.Profinet_PLC_OUTPUTS[2].0:= P1_Robot.KOM_OUT.PolozDPS_4F_na_PowerCP;
	P1_Robot.KOM_OUT.Profinet_PLC_OUTPUTS[2].1:= P1_Robot.KOM_OUT.PolozDPS_5F_na_PowerCP;
	P1_Robot.KOM_OUT.Profinet_PLC_OUTPUTS[2].2:= P1_Robot.KOM_OUT.PolozFoam4F_na_PowerCP;
	P1_Robot.KOM_OUT.Profinet_PLC_OUTPUTS[2].3:= P1_Robot.KOM_OUT.PolozFoam5F_na_PowerCP;
	P1_Robot.KOM_OUT.Profinet_PLC_OUTPUTS[2].4:= P1_Robot.KOM_OUT.PolozSpodnyBusbar4F_na_PowerCP;
	P1_Robot.KOM_OUT.Profinet_PLC_OUTPUTS[2].5:= P1_Robot.KOM_OUT.PolozSpodnyBusbar5F_na_PowerCP;
	P1_Robot.KOM_OUT.Profinet_PLC_OUTPUTS[2].6:= P1_Robot.KOM_OUT.PolozSpodnyBusbar5H_na_PowerCP;
	P1_Robot.KOM_OUT.Profinet_PLC_OUTPUTS[2].7:= P1_Robot.KOM_OUT.Presun_CakaciaPozicia;

	P1_Robot.KOM_OUT.Profinet_PLC_OUTPUTS[3].0:= P1_Robot.IN.DokStanPritGrip_BusBary5H_IS77;
	P1_Robot.KOM_OUT.Profinet_PLC_OUTPUTS[3].1:= P1_Robot.IN.DokStanPritGrip_BusBary45F_IS78;
	P1_Robot.KOM_OUT.Profinet_PLC_OUTPUTS[3].2:= P1_Robot.IN.Griper_Otvoreny_MS40;
	P1_Robot.KOM_OUT.Profinet_PLC_OUTPUTS[3].3:= P1_Robot.IN.Griper_Zatvoreny_MS41;
	P1_Robot.KOM_OUT.Profinet_PLC_OUTPUTS[3].4:= P1_Robot.IN.SnimacVakua_S20;
	P1_Robot.KOM_OUT.Profinet_PLC_OUTPUTS[3].5:= P1_Robot.KOM_OUT.TypGripra_45F;
	P1_Robot.KOM_OUT.Profinet_PLC_OUTPUTS[3].6:= P1_Robot.KOM_OUT.TypGripra_5H;
    P1_Robot.KOM_OUT.Profinet_PLC_OUTPUTS[3].7:= P1_Robot.KOM_OUT.Odparkovanie;

    P1_Robot.KOM_OUT.Profinet_PLC_OUTPUTS[4].0:= P1_Robot.KOM_OUT.UvolniBusbary;
	P1_Robot.KOM_OUT.Profinet_PLC_OUTPUTS[4].1:= P1_Robot.KOM_OUT.ZopakujOdoberanie;

END_ACTION
```

### Program Logical/Program/Pracovisko_1/P1_OvladanieVizu (IEC)

#### Main.st - Init, cyclic, exit code
```iecst
PROGRAM _INIT
	P1_Vizu.GoPage:= 'PageBootP1';

END_PROGRAM

PROGRAM _CYCLIC

	//************************************Filter alarmov**************************************************************//
	FilterVizu_P1:= '[{"logicalOperator":"and","value":100,"conditionType":">=","columnType":"cod","useAlarmState":false,"alarmState":0},{"value":199,"conditionType":"<=","columnType":"cod","useAlarmState":false,"alarmState":0}]';

	//***********************************Zobrazenie warningov pracoviska****************************************************//
	//0 - Pracovisko je vypnuté.
	//1 - Prebieha inicializácia pracoviska.
	//2 - Na pracovisku prebieha výroba.
	//3 - Prebieha ukončenie pracovného cyklu pracoviska.
	//4 - Prebieha režim vyprázdnenia linky.
	//5 - Robot nie je prepnuty do automatického režimu !!!
	//6 - Doplň zásobník skrutiek K30 !!!
	//7 - Doplň zásobník skrutiek M5 !!!
    //8 - Doplň zásobník skrutiek M4 !!!
    //10 - Testovací kus

	IF NOT P1_Robot.KOM_IN.Stav_RezimAUTOMAT THEN
		P1_Vizu.Warnings_Index:= 5;
	ELSIF P1_Srobovanie.STAV.Zasobnik_K30_Prazdny THEN
		P1_Vizu.Warnings_Index:= 6;
	ELSIF P1_Srobovanie.STAV.Zasobnik_M5_Prazdny THEN
		P1_Vizu.Warnings_Index:= 7;
	ELSIF P1_Srobovanie.STAV.Zasobnik_M4_Prazdny THEN
        P1_Vizu.Warnings_Index:= 8;
    ELSIF Linka.TestovaciKus THEN
        P1_Vizu.Warnings_Index:= 10;
	ELSIF Linka.VyprazdnenieLinky THEN
		P1_Vizu.Warnings_Index:= 4;
	ELSIF P1_Pracovisko.STAV.Automat AND NOT P1_Pracovisko.STAV.PoINIT AND NOT P1_Pracovisko.STAV.UkoncenieCyklu_BUSY THEN
		P1_Vizu.Warnings_Index:= 1;
	ELSIF P1_Pracovisko.STAV.PoINIT AND NOT P1_Pracovisko.STAV.UkoncenieCyklu_BUSY THEN
		P1_Vizu.Warnings_Index:= 2;
	ELSIF P1_Pracovisko.STAV.UkoncenieCyklu_BUSY THEN
		P1_Vizu.Warnings_Index:= 3;
	ELSIF NOT P1_Pracovisko.STAV.Automat THEN
		P1_Vizu.Warnings_Index:= 0;
	END_IF

		//************************Prepínanie farby textového pola warning zariadenia***********************************//
		IF P1_Vizu.Warnings_Index = 0 THEN
			P1_Vizu.Warnings_Farba:= "TextOutput_Green";
	ELSIF P1_Vizu.Warnings_Index = 1 THEN
		P1_Vizu.Warnings_Farba:= "TextOutput_Green";
	ELSIF P1_Vizu.Warnings_Index = 2 THEN
		P1_Vizu.Warnings_Farba:= "TextOutput_Green";
	ELSIF P1_Vizu.Warnings_Index = 3 THEN
		P1_Vizu.Warnings_Farba:= "TextOutput_Green";
	ELSIF P1_Vizu.Warnings_Index = 4 THEN
        P1_Vizu.Warnings_Farba:= "TextOutput_Green";
    ELSIF P1_Vizu.Warnings_Index = 10 THEN
        P1_Vizu.Warnings_Farba:= "TextOutput_Green";
	ELSE
		IF Blikac1s THEN
			P1_Vizu.Warnings_Farba:= "TextOutput_Red";
		ELSE
			P1_Vizu.Warnings_Farba:= "TextOutput_Grey";
		END_IF
	END_IF

	//***********************Prepnutie na obrazovku Automat z ručného režimu******************//
    IF P1_Pracovisko.STAV.Manual AND NOT Safety.STAV.P1_ZamkyBunky_AKTIVNE THEN
        P1_Pracovisko.Reset:= TRUE;
        P1_Vizu.GoPage:= 'PageBootP1';
    END_IF

	//***********************Prepnutie bootovacej obrazovky********************************//
	IF NOT Safety.STAV.SafetyPLC_Nabehlo THEN
        P1_Vizu.GoPage:= 'PageBootP1';
    ELSIF CasPrepnutiaObrazovky.Q THEN
        P1_Vizu.GoPage:= 'PageBootP1';
	ELSIF P1_Vizu.ActualPage = 'PageBootP1' AND Safety.STAV.SafetyPLC_Nabehlo THEN
		P1_Vizu.GoPage:= 'PageAutomatP1';
	END_IF

    CasPrepnutiaObrazovky.IN:= P1_Vizu.ActualPage = 'PageBootP1' AND P1_Vizu.GoPage = 'PageAutomatP1';
    CasPrepnutiaObrazovky.PT:= T#5s;
    CasPrepnutiaObrazovky();

	//*************************************Zamknutie tlačítok***************************************************************//
	//Tlačítko Štat Automat//
	IF P1_Pracovisko.STAV.UkoncenieCyklu_BUSY THEN
        P1_Vizu.TL_StartAutomat_ENABLE:= FALSE;
    ELSIF P1_Pracovisko.STAV.PORUCHA THEN
        P1_Vizu.TL_StartAutomat_ENABLE:= FALSE;
    ELSIF NOT P1_Robot.KOM_IN.Stav_RezimAUTOMAT THEN
		P1_Vizu.TL_StartAutomat_ENABLE:= FALSE;
	ELSIF NOT Safety.STAV.P1_ZonaBunky_AKTIVNA THEN
		P1_Vizu.TL_StartAutomat_ENABLE:= FALSE;
	ELSE
        P1_Vizu.TL_StartAutomat_ENABLE:= TRUE;
    END_IF

    //Tlačítko Ukončenie Cyklu//
	IF P1_Pracovisko.STAV.PoINIT THEN
		P1_Vizu.TL_KoniecCyklu_ENABLE:= TRUE;
	ELSE
		P1_Vizu.TL_KoniecCyklu_ENABLE:= FALSE;
	END_IF

    //Tlačítko STOP//
    IF P1_Pracovisko.STAV.PoINIT THEN
        P1_Vizu.TL_STOP_ENABLE:= FALSE;
    ELSE
        P1_Vizu.TL_STOP_ENABLE:= TRUE;
    END_IF

	//Tlačítko Režim Automat//

    P1_Vizu.TL_RezimAutomat_ENABLE:= TRUE;

	//Tlačítko Režim Manual//
	IF P1_Pracovisko.STAV.Automat THEN
		P1_Vizu.TL_RezimManual_ENABLE:= FALSE;
	ELSIF NOT P1_Pracovisko.STAV.Manual AND NOT P1_Pracovisko.STAV.READY THEN
        P1_Vizu.TL_RezimManual_ENABLE:= FALSE;
    ELSIF NOT Safety.STAV.P1_ZamkyBunky_AKTIVNE THEN
        P1_Vizu.TL_RezimManual_ENABLE:= FALSE;
	ELSE
		P1_Vizu.TL_RezimManual_ENABLE:= TRUE;
	END_IF

	//Tlačítka ovládania zámkov//
	IF NOT P1_Pracovisko.STAV.Automat THEN
		P1_Vizu.TL_OvladaniaZamkov_ENABLE:= TRUE;
	ELSE
		P1_Vizu.TL_OvladaniaZamkov_ENABLE:= FALSE;
	END_IF

    //Tlačítko zmena modelu//
    IF Linka.STAV.Vypnuta THEN
        P1_Vizu.TL_VolbaModelu_ENABLE:= TRUE;
    ELSE
        P1_Vizu.TL_VolbaModelu_ENABLE:= FALSE;
    END_IF

	//Tlačítko paletka prechádza//
    IF NOT Linka.STAV.PoINIT THEN
        P1_Vizu.TL_PaletkaPrechadza_ENABLE:= FALSE;
    ELSIF NOT P1_Vytah.IN.PritomnostPaletky_S19 THEN
        P1_Vizu.TL_PaletkaPrechadza_ENABLE:= FALSE;
    ELSIF Linka.TestovaciKus THEN
        P1_Vizu.TL_PaletkaPrechadza_ENABLE:= FALSE;
    ELSIF Linka.Revork THEN
        P1_Vizu.TL_PaletkaPrechadza_ENABLE:= FALSE;
    ELSIF Linka.PaletkaPrechadza THEN
        P1_Vizu.TL_PaletkaPrechadza_ENABLE:= FALSE;
    ELSE
        P1_Vizu.TL_PaletkaPrechadza_ENABLE:= TRUE;
    END_IF

	//Tlačítko vyprázdnenie linky//
	IF Linka.VyprazdnenieLinky THEN
		P1_Vizu.TL_VyprazdnenieLinky_ENABLE:= FALSE;
	ELSIF NOT P4_Pracovisko.STAV.Automat THEN
        P1_Vizu.TL_VyprazdnenieLinky_ENABLE:= FALSE;
    ELSIF Linka.TestovaciKus THEN
        P1_Vizu.TL_VyprazdnenieLinky_ENABLE:= FALSE;
    ELSE
		P1_Vizu.TL_VyprazdnenieLinky_ENABLE:= TRUE;
	END_IF

    //Tlačítko testovací kus//
    IF NOT Linka.STAV.PoINIT THEN
        P1_Vizu.TL_TestovaciKus_ENABLE:= FALSE;
    ELSIF Linka.Revork THEN
        P1_Vizu.TL_TestovaciKus_ENABLE:= FALSE;
    ELSIF NOT P1_Vytah.IN.PritomnostPaletky_S19 THEN
        P1_Vizu.TL_TestovaciKus_ENABLE:= FALSE;
    ELSIF Linka.PaletkaPrechadza THEN
        P1_Vizu.TL_TestovaciKus_ENABLE:= FALSE;
    ELSE
        P1_Vizu.TL_TestovaciKus_ENABLE:= TRUE;
    END_IF

    //Tlačítko retest//
    IF NOT Linka.STAV.PoINIT THEN
        P1_Vizu.TL_Revork_ENABLE:= FALSE;
    ELSIF NOT P1_Vytah.IN.PritomnostPaletky_S19 THEN
        P1_Vizu.TL_Revork_ENABLE:= FALSE;
    ELSIF Linka.TestovaciKus THEN
        P1_Vizu.TL_Revork_ENABLE:= FALSE;
    ELSIF Linka.PaletkaPrechadza THEN
        P1_Vizu.TL_Revork_ENABLE:= FALSE;
    ELSE
        P1_Vizu.TL_Revork_ENABLE:= TRUE;
    END_IF

    //Tlačítka spustenie čistenie skrutkovačiek v ručnom režime//
    IF NOT P1_Srobovacky_VychodziaPozicia THEN
        P1_Vizu.RR_CistenieSkrutkovaciek_ENABLE:= FALSE;
    ELSIF P1_Srobovanie.STAV.Cistenie_M4_BUSY THEN
        P1_Vizu.RR_CistenieSkrutkovaciek_ENABLE:= FALSE;
    ELSIF P1_Srobovanie.STAV.Cistenie_K30_BUSY THEN
        P1_Vizu.RR_CistenieSkrutkovaciek_ENABLE:= FALSE;
    ELSIF NOT P1_Srobovanie.STAV.OsX_HomingOK THEN
        P1_Vizu.RR_CistenieSkrutkovaciek_ENABLE:= FALSE;
    ELSIF NOT P1_Srobovanie.STAV.OsY_HomingOK THEN
        P1_Vizu.RR_CistenieSkrutkovaciek_ENABLE:= FALSE;
    ELSE
        P1_Vizu.RR_CistenieSkrutkovaciek_ENABLE:= TRUE;
    END_IF

    //Tlačítka ovládania výťahu v ručnom režime//
    IF NOT P1_Vytah.STAV.ServoZdvihu_HomingOK THEN
        P1_Vizu.TL_OvladanieVytahu_ENABLE:= FALSE;
    ELSIF P1_Vytah.STAV.ServoZdvihu_Homing_BUSY THEN
        P1_Vizu.TL_OvladanieVytahu_ENABLE:= FALSE;
    ELSIF P1_Vytah.IN.VystupDopravnikaVytahu_OS12 THEN
        P1_Vizu.TL_OvladanieVytahu_ENABLE:= FALSE;
    ELSIF NOT Safety.STAV.P1_Vytah_Bariera_AKTIVNA THEN
        P1_Vizu.TL_OvladanieVytahu_ENABLE:= FALSE;
    ELSE
        P1_Vizu.TL_OvladanieVytahu_ENABLE:= TRUE;
    END_IF

    //Tlačítko homing zdvihu výťahu//
    IF P1_Vytah.IN.VystupDopravnikaVytahu_OS12 THEN
        P1_Vizu.TL_HomingVytahu_ENABLE:= FALSE;
    ELSIF NOT Safety.STAV.P1_Vytah_Bariera_AKTIVNA THEN
       P1_Vizu.TL_HomingVytahu_ENABLE:= FALSE;
    ELSE
        P1_Vizu.TL_HomingVytahu_ENABLE:= TRUE;
    END_IF

    //Tlačítka ovládanie osy X manipulátora šróbovačiek//
    IF NOT P1_Srobovanie.STAV.OsX_HomingOK THEN
        P1_Vizu.Srobovanie_OvlManipOsX_ENABLE:= FALSE;
    ELSIF NOT P1_Srobovacky_VychodziaPozicia THEN
        P1_Vizu.Srobovanie_OvlManipOsX_ENABLE:= FALSE;
    ELSIF P1_Srobovanie.RR_PolohujNaPoziciuSkrutky_4F THEN
        P1_Vizu.Srobovanie_OvlManipOsX_ENABLE:= FALSE;
    ELSIF P1_Srobovanie.RR_PolohujNaPoziciuSkrutky_5F THEN
        P1_Vizu.Srobovanie_OvlManipOsX_ENABLE:= FALSE;
    ELSIF P1_Srobovanie.RR_PolohujNaPoziciuSkrutky_5H THEN
        P1_Vizu.Srobovanie_OvlManipOsX_ENABLE:= FALSE;
    ELSIF P1_Srobovanie.STAV.Cistenie_K30_BUSY THEN
        P1_Vizu.Srobovanie_OvlManipOsX_ENABLE:= FALSE;
    ELSIF P1_Srobovanie.STAV.Cistenie_M4_BUSY THEN
        P1_Vizu.Srobovanie_OvlManipOsX_ENABLE:= FALSE;
    ELSE
        P1_Vizu.Srobovanie_OvlManipOsX_ENABLE:= TRUE;
    END_IF

    //Tlačítka ovládania osy Y manipulatora šróbovačiek//
    IF NOT P1_Srobovanie.STAV.OsY_HomingOK THEN
        P1_Vizu.Srobovanie_OvlManipOsY_ENABLE:= FALSE;
    ELSIF NOT P1_Srobovacky_VychodziaPozicia THEN
        P1_Vizu.Srobovanie_OvlManipOsY_ENABLE:= FALSE;
    ELSIF P1_Srobovanie.RR_PolohujNaPoziciuSkrutky_4F THEN
        P1_Vizu.Srobovanie_OvlManipOsY_ENABLE:= FALSE;
    ELSIF P1_Srobovanie.RR_PolohujNaPoziciuSkrutky_5F THEN
        P1_Vizu.Srobovanie_OvlManipOsY_ENABLE:= FALSE;
    ELSIF P1_Srobovanie.RR_PolohujNaPoziciuSkrutky_5H THEN
        P1_Vizu.Srobovanie_OvlManipOsY_ENABLE:= FALSE;
    ELSIF P1_Srobovanie.STAV.Cistenie_K30_BUSY THEN
        P1_Vizu.Srobovanie_OvlManipOsY_ENABLE:= FALSE;
    ELSIF P1_Srobovanie.STAV.Cistenie_M4_BUSY THEN
        P1_Vizu.Srobovanie_OvlManipOsY_ENABLE:= FALSE;
    ELSE
        P1_Vizu.Srobovanie_OvlManipOsY_ENABLE:= TRUE;
    END_IF

    //Tlačítka spustenie čistenie skrutkovačiek v ručnom režime//
    IF NOT P1_Srobovacky_VychodziaPozicia THEN
        P1_Vizu.RR_CistenieSkrutkovaciek_ENABLE:= FALSE;
    ELSIF P1_Srobovanie.STAV.Cistenie_K30_BUSY THEN
        P1_Vizu.RR_CistenieSkrutkovaciek_ENABLE:= FALSE;
    ELSIF P1_Srobovanie.STAV.Cistenie_M4_BUSY THEN
        P1_Vizu.RR_CistenieSkrutkovaciek_ENABLE:= FALSE;
    ELSIF NOT P1_Srobovanie.STAV.OsX_HomingOK THEN
        P1_Vizu.RR_CistenieSkrutkovaciek_ENABLE:= FALSE;
    ELSIF NOT P1_Srobovanie.STAV.OsY_HomingOK THEN
        P1_Vizu.RR_CistenieSkrutkovaciek_ENABLE:= FALSE;
    ELSIF P1_UrovenPrihlasenehoUzivatela < 20 THEN
        P1_Vizu.RR_CistenieSkrutkovaciek_ENABLE:= FALSE;
    ELSIF P1_Srobovanie.RR_PolohujNaPoziciuSkrutky_4F THEN
        P1_Vizu.RR_CistenieSkrutkovaciek_ENABLE:= FALSE;
    ELSIF P1_Srobovanie.RR_PolohujNaPoziciuSkrutky_5F THEN
        P1_Vizu.RR_CistenieSkrutkovaciek_ENABLE:= FALSE;
    ELSIF P1_Srobovanie.RR_PolohujNaPoziciuSkrutky_5H THEN
        P1_Vizu.RR_CistenieSkrutkovaciek_ENABLE:= FALSE;
    ELSE
        P1_Vizu.RR_CistenieSkrutkovaciek_ENABLE:= TRUE;
    END_IF

    //Tlačítko editácie uživatelov//
    IF P1_UrovenPrihlasenehoUzivatela = 100 THEN
        P1_Vizu.TL_Uzivatelia_ENABLE:= TRUE;
    ELSE
        P1_Vizu.TL_Uzivatelia_ENABLE:= FALSE;
    END_IF

    //Zamknutie tlačítok test pozicii skrutkovačiek//
    IF NOT P1_Srobovanie.STAV.OsX_HomingOK THEN
        P1_Vizu.RR_PozicieSkrutiek_ENABLE:= FALSE;
    ELSIF NOT P1_Srobovanie.STAV.OsY_HomingOK THEN
        P1_Vizu.RR_PozicieSkrutiek_ENABLE:= FALSE;
    ELSIF NOT P1_Srobovacky_VychodziaPozicia THEN
        P1_Vizu.RR_PozicieSkrutiek_ENABLE:= FALSE;
    ELSIF P1_Srobovanie.STAV.Cistenie_K30_BUSY THEN
        P1_Vizu.RR_PozicieSkrutiek_ENABLE:= FALSE;
    ELSIF P1_Srobovanie.STAV.Cistenie_M4_BUSY THEN
        P1_Vizu.RR_PozicieSkrutiek_ENABLE:= FALSE;
    ELSIF P1_UrovenPrihlasenehoUzivatela < 100 THEN
        P1_Vizu.RR_PozicieSkrutiek_ENABLE:= FALSE;
    ELSIF P1_Srobovanie.RR_PolohujNaPoziciuSkrutky_4F THEN
        P1_Vizu.RR_PozicieSkrutiek_ENABLE:= FALSE;
    ELSIF P1_Srobovanie.RR_PolohujNaPoziciuSkrutky_5F THEN
        P1_Vizu.RR_PozicieSkrutiek_ENABLE:= FALSE;
    ELSIF P1_Srobovanie.RR_PolohujNaPoziciuSkrutky_5H THEN
        P1_Vizu.RR_PozicieSkrutiek_ENABLE:= FALSE;
    ELSE
        P1_Vizu.RR_PozicieSkrutiek_ENABLE:= TRUE;
    END_IF

    //**************************Zamknutie editácie parametrov*********************************//
   IF P1_UrovenPrihlasenehoUzivatela >= 20 THEN
        P1_Vizu.EditaciaParametrov_ENABLE:= TRUE;
   ELSE
        P1_Vizu.EditaciaParametrov_ENABLE:= FALSE;
   END_IF

	//***************************************Zmena farieb tlačítok pre ovládanie zámkou********************************//
	//Predné dvere //
	IF Safety.OUT.P1_ZamkniZamok_PredneDvere AND Safety.IN.P1_PredneDvere_PritomPetlice THEN
		P1_Vizu.TL_PrednyZamok_Farba:= "Button_Green";
	ELSIF Safety.IN.P1_PredneDvere_PritomPetlice THEN
		IF Blikac1s THEN
			P1_Vizu.TL_PrednyZamok_Farba:= "Button_Blue";
		ELSE
			P1_Vizu.TL_PrednyZamok_Farba:= "Operate";
		END_IF
	ELSE
		P1_Vizu.TL_PrednyZamok_Farba:= "Button_Red";
	END_IF

	//Zadné dvere pravá strana//
	IF Safety.OUT.P1_ZamkniZamok_ZadneDverePS AND Safety.IN.P1_ZadneDverePS_PritomPetlice THEN
		P1_Vizu.TL_ZadnyZamokPS_Farba:= "Button_Green";
	ELSIF Safety.IN.P1_ZadneDverePS_PritomPetlice THEN
		IF Blikac1s THEN
			P1_Vizu.TL_ZadnyZamokPS_Farba:= "Button_Blue";
		ELSE
			P1_Vizu.TL_ZadnyZamokPS_Farba:= "Operate";
		END_IF
	ELSE
		P1_Vizu.TL_ZadnyZamokPS_Farba:= "Button_Red";
	END_IF

	//Zadné dvere lavá strana//
	IF Safety.OUT.P1_ZamkniZamok_ZadneDvereLS AND Safety.IN.P1_ZadneDvereLS_PritomPetlice THEN
		P1_Vizu.TL_ZadnyZamokLS_Farba:= "Button_Green";
	ELSIF Safety.IN.P1_ZadneDvereLS_PritomPetlice THEN
		IF Blikac1s THEN
			P1_Vizu.TL_ZadnyZamokLS_Farba:= "Button_Blue";
		ELSE
			P1_Vizu.TL_ZadnyZamokLS_Farba:= "Operate";
		END_IF
	ELSE
		P1_Vizu.TL_ZadnyZamokLS_Farba:= "Button_Red";
	END_IF

	//***********************************Prepínanie stavov pracovísk*******************************************************************//
	//Výťah//
	IF NOT P1_Vytah.IN.Dopravnik_READY THEN
		P1_Vizu.IndexStavu_Vytah:= 3;
	ELSIF P1_PoruchaST1 THEN
		P1_Vizu.IndexStavu_Vytah:= 3;
	ELSIF P1_Vytah.Automat AND NOT P1_Vytah.STAV.PoINIT THEN
		P1_Vizu.IndexStavu_Vytah:= 1;
	ELSIF P1_Vytah.Automat AND P1_Vytah.STAV.PoINIT THEN
		P1_Vizu.IndexStavu_Vytah:= 2;
	ELSE
		P1_Vizu.IndexStavu_Vytah:= 0;
	END_IF

	//Dopravníky//
	IF NOT P1_Dopravniky.IN.HornyDoprav_READY OR NOT P1_Dopravniky.IN.SpodnyDoprav_READY THEN
		P1_Vizu.IndexStavu_Dopravnik:= 3;
	ELSIF P1_Dopravniky.Automat AND NOT P1_Dopravniky.STAV.PoINIT THEN
		P1_Vizu.IndexStavu_Dopravnik:= 1;
	ELSIF P1_Dopravniky.Automat AND P1_Dopravniky.STAV.PoINIT THEN
		P1_Vizu.IndexStavu_Dopravnik:= 2;
	ELSE
		P1_Vizu.IndexStavu_Dopravnik:= 0;
	END_IF

	//Spodný stoper//
	IF P1_SpodnyStoper.Automat AND NOT P1_SpodnyStoper.STAV.PoINIT THEN
		P1_Vizu.IndexStavu_SpodnyStoper:= 1;
	ELSIF P1_SpodnyStoper.Automat AND P1_SpodnyStoper.STAV.PoINIT THEN
		P1_Vizu.IndexStavu_SpodnyStoper:= 2;
	ELSE
		P1_Vizu.IndexStavu_SpodnyStoper:= 0;
	END_IF

	//Stoper šrobovania//
	IF P1_PoruchaST2 THEN
		P1_Vizu.IndexStavu_StoperSrobovania:= 3;
	ELSIF P1_StoperSrobovania.Automat AND NOT P1_StoperSrobovania.STAV.PoINIT THEN
		P1_Vizu.IndexStavu_StoperSrobovania:= 1;
	ELSIF P1_StoperSrobovania.Automat AND P1_StoperSrobovania.STAV.PoINIT THEN
		P1_Vizu.IndexStavu_StoperSrobovania:= 2;
	ELSE
		P1_Vizu.IndexStavu_StoperSrobovania:= 0;
	END_IF

	//Šrobovanie//
	IF P1_PoruchaST2 THEN
		P1_Vizu.IndexStavu_Srobovanie:= 3;
	ELSIF P1_Srobovanie.Automat AND NOT P1_Srobovanie.STAV.PoINIT THEN
		P1_Vizu.IndexStavu_Srobovanie:= 1;
	ELSIF P1_Srobovanie.Automat AND P1_Srobovanie.STAV.PoINIT THEN
		P1_Vizu.IndexStavu_Srobovanie:= 2;
	ELSE
		P1_Vizu.IndexStavu_Srobovanie:= 0;
	END_IF

	//Akumulačný stoper//
	IF P1_AkumulacnyStoper.Automat AND NOT P1_AkumulacnyStoper.STAV.PoINIT THEN
		P1_Vizu.IndexStavu_AkumulacnyStoper:= 1;
	ELSIF P1_AkumulacnyStoper.Automat AND P1_AkumulacnyStoper.STAV.PoINIT THEN
		P1_Vizu.IndexStavu_AkumulacnyStoper:= 2;
	ELSE
		P1_Vizu.IndexStavu_AkumulacnyStoper:= 0;
	END_IF

	//Robot//
	IF P1_Robot.Automat AND NOT P1_Robot.STAV.PoINIT THEN
		P1_Vizu.IndexStavu_Robot:= 1;
	ELSIF P1_Robot.Automat AND P1_Robot.STAV.PoINIT THEN
		P1_Vizu.IndexStavu_Robot:= 2;
	ELSE
		P1_Vizu.IndexStavu_Robot:= 0;
	END_IF

END_PROGRAM

PROGRAM _EXIT
	(* Insert code here *)

END_PROGRAM
```

#### Variables.var - Local variables
```iecst
VAR
	CasPrepnutiaObrazovky : TON;
END_VAR
```

### Program Logical/Program/Pracovisko_1/P1_OvladanieSafety (IEC)

#### Main.st - Init, cyclic, exit code
```iecst
PROGRAM _INIT
	(* Insert code here *)

END_PROGRAM

PROGRAM _CYCLIC

	//******************************************Ovládanie zámkov dverí bunky****************************************//
	//Predné dvere //
	IF EDGEPOS(P1_Vizu.TL_ZamkniPrednyZamok) THEN
		IF NOT Safety.OUT.P1_ZamkniZamok_PredneDvere AND Safety.IN.P1_PredneDvere_PritomPetlice THEN
			Safety.OUT.P1_ZamkniZamok_PredneDvere:= TRUE;
		ELSIF Safety.OUT.P1_ZamkniZamok_PredneDvere THEN
			Safety.OUT.P1_ZamkniZamok_PredneDvere:= FALSE;
		END_IF
		P1_Vizu.TL_ZamkniPrednyZamok:= FALSE;
	END_IF

	//Zadné dvere - pravá strana//
	IF EDGEPOS(P1_Vizu.TL_ZamkniZadnyZamokPS) THEN
		IF NOT Safety.OUT.P1_ZamkniZamok_ZadneDverePS AND Safety.IN.P1_ZadneDverePS_PritomPetlice THEN
			Safety.OUT.P1_ZamkniZamok_ZadneDverePS:= TRUE;
		ELSIF Safety.OUT.P1_ZamkniZamok_ZadneDverePS THEN
			Safety.OUT.P1_ZamkniZamok_ZadneDverePS:= FALSE;
		END_IF
		P1_Vizu.TL_ZamkniZadnyZamokPS:= FALSE;
	END_IF

	//Zadné dvere - lavá strana//
	IF EDGEPOS(P1_Vizu.TL_ZamkniZadnyZamokLS) THEN
		IF NOT Safety.OUT.P1_ZamkniZamok_ZadneDvereLS AND Safety.IN.P1_ZadneDvereLS_PritomPetlice THEN
			Safety.OUT.P1_ZamkniZamok_ZadneDvereLS:= TRUE;
		ELSIF Safety.OUT.P1_ZamkniZamok_ZadneDvereLS THEN
			Safety.OUT.P1_ZamkniZamok_ZadneDvereLS:= FALSE;
		END_IF
		P1_Vizu.TL_ZamkniZadnyZamokLS:= FALSE;
	END_IF

	//Reset zóny Výtahu//
	CasResetZonyVytahu.IN:= NOT Safety.STAV.P1_ZonaVytahu_AKTIVNA AND Safety.STAV.ZonaCS_AKTIVNA AND (Safety.STAV.P1_Vytah_Bariera_AKTIVNA OR Safety.STAV.P1_SnimacVytahu_AKTIVNY);

	IF CasResetZonyVytahu.Q THEN
		Safety.IN.P1_ZonaVytahu_RESET:= TRUE;
	ELSE
		Safety.IN.P1_ZonaVytahu_RESET:= FALSE;
	END_IF

	CasResetZonyVytahu.PT:= T#1s;
	CasResetZonyVytahu();

	//Reset zóny bunky//
	CasResetZonyBunky.IN:= NOT Safety.STAV.P1_ZonaBunky_AKTIVNA	AND Safety.STAV.ZonaCS_AKTIVNA AND Safety.STAV.P1_ZamkyBunky_AKTIVNE AND (Safety.STAV.P1_VstupBunky_Bariera_AKTIVNA OR Safety.STAV.P1_VystupTunela_Bariera_AKTIVNA);

	IF CasResetZonyBunky.Q THEN
		Safety.IN.P1_ZonaBunky_RESET:= TRUE;
	ELSE
		Safety.IN.P1_ZonaBunky_RESET:= FALSE;
	END_IF

	CasResetZonyBunky.PT:= T#1s;
	CasResetZonyBunky();

END_PROGRAM

PROGRAM _EXIT
	(* Insert code here *)

END_PROGRAM
```

#### Variables.var - Local variables
```iecst
VAR
	CasResetZonyVytahu : TON;
	CasResetZonyBunky : TON;
END_VAR
```

### Program Logical/Program/Pracovisko_1/P1_Vytah (IEC)
